{attribute 'global_init_slot' := '40510'}
VAR_GLOBAL
  LblPlt_Facade                                            :FB_BA_Label:=( sObjName:='FAS', sDescr:='Fassade');
  LblPlt_Natural_smoke_extraction                          :FB_BA_Label:=( sObjName:='NRA', sDescr:='Natürlicher Rauchabzug');
  LblPlt_Doors_gates_sluices                               :FB_BA_Label:=( sObjName:='TUE', sDescr:='Türen, Tore, Schleusen');
  LblPlt_Smoke_and_heat_extraction_system                  :FB_BA_Label:=( sObjName:='RWA', sDescr:='Rauch- und Wärmeabzugsanlage');
  LblPlt_Sunlight_protection                               :FB_BA_Label:=( sObjName:='SON', sDescr:='Sonnenschutzanlage');
// 411 Abwasseranlagen
  LblPlt_Separator_facility                                :FB_BA_Label:=( sObjName:='ABS', sDescr:='Abscheideranlage');
  LblPlt_Lifting_system                                    :FB_BA_Label:=( sObjName:='HBA', sDescr:='Hebeanlage');
  LblPlt_Neutralisation_plant                              :FB_BA_Label:=( sObjName:='NEU', sDescr:='Neutralisationsanlage');
// 412 Wasseranlagen
  LblPlt_Trace_heating                                     :FB_BA_Label:=( sObjName:='BGH', sDescr:='Begleitheizung');
  LblPlt_Process_water                                     :FB_BA_Label:=( sObjName:='BTW', sDescr:='Betriebswasser');
  LblPlt_Well_water                                        :FB_BA_Label:=( sObjName:='BWA', sDescr:='Brunnenwasser');
  LblPlt_Dispensing_installation                           :FB_BA_Label:=( sObjName:='DOS', sDescr:='Dosieranlage');
  LblPlt_Pressure_booster_system                           :FB_BA_Label:=( sObjName:='DEA', sDescr:='Druckerhöhungsanlage');
  LblPlt_Softening_unit                                    :FB_BA_Label:=( sObjName:='EHA', sDescr:='Enthärtungsanlage');
// Trinkwasser
  LblPlt_Drinking_water_heating_system                     :FB_BA_Label:=( sObjName:='TWE', sDescr:='Trinkwassererwärmungsanlage');
  LblPlt_Reverse_osmosis_system                            :FB_BA_Label:=( sObjName:='UKO', sDescr:='Umkehrosmoseanlage');
  LblPlt_Desalination_plant                                :FB_BA_Label:=( sObjName:='VEA', sDescr:='Vollentsalzungsanlage');
// 421 Wärmeerzeugungsanlagen
  LblPlt_BHKW                                              :FB_BA_Label:=( sObjName:='BHK', sDescr:='BHKW');
  LblPlt_Electric_heating                                  :FB_BA_Label:=( sObjName:='EHZ', sDescr:='Elektroheizung');
  LblPlt_District_heating_transfer                         :FB_BA_Label:=( sObjName:='FWÜ', sDescr:='Fernwärmeübergabe');
// Geothermieanlage
  LblPlt_Boiler                                            :FB_BA_Label:=( sObjName:='KES', sDescr:='Kessel');
  LblPlt_Clean_steam_generation                            :FB_BA_Label:=( sObjName:='RDE', sDescr:='Reindampferzeugung');
  LblPlt_Solar_power_system                                :FB_BA_Label:=( sObjName:='SOL', sDescr:='Solaranlage');
  LblPlt_Heating_pump                                      :FB_BA_Label:=( sObjName:='WPU', sDescr:='Wärmepumpe');
// 422 Wärmeverteilnetze
  LblPlt_Pressure_maintenance                              :FB_BA_Label:=( sObjName:='DHG', sDescr:='Druckhaltung');
  LblPlt_Heating_circuit                                   :FB_BA_Label:=( sObjName:='HZK', sDescr:='Heizkreis');
  LblPlt_Heating                                           :FB_BA_Label:=( sObjName:='HZG', sDescr:='Heizung');
  LblPlt_Back_feed_system                                  :FB_BA_Label:=( sObjName:='NSA', sDescr:='Nachspeiseanlage');
  LblPlt_Buffer                                            :FB_BA_Label:=( sObjName:='PFS', sDescr:='Pufferspeicher');
  LblPlt_Heat_distribution_network                         :FB_BA_Label:=( sObjName:='WVN', sDescr:='Wärmeverteilnetz');
  LblPlt_Heat_exchanger                                    :FB_BA_Label:=( sObjName:='WTR', sDescr:='Wärmeüberträger');
// 423 Raumheizflächen
  LblPlt_Concrete_core_activation                          :FB_BA_Label:=( sObjName:='BKA', sDescr:='Betonkernaktivierung');
  LblPlt_Overhead_heating                                  :FB_BA_Label:=( sObjName:='DHZ', sDescr:='Deckenheizung');
  LblPlt_Ceiling_radiator_panels                           :FB_BA_Label:=( sObjName:='DSP', sDescr:='Deckenstrahlplatten');
  LblPlt_Facade_heating                                    :FB_BA_Label:=( sObjName:='FAH', sDescr:='Fassadenheizung');
  LblPlt_Panel_heating                                     :FB_BA_Label:=( sObjName:='FLH', sDescr:='Flächenheizung');
  LblPlt_Underfloor_heating                                :FB_BA_Label:=( sObjName:='FBH', sDescr:='Fußbodenheizung');
  LblPlt_Heated_chilled_ceiling                            :FB_BA_Label:=( sObjName:='HKD', sDescr:='Heiz-/Kühldecke');
  LblPlt_Static_heating                                    :FB_BA_Label:=( sObjName:='STH', sDescr:='Statische Heizung');
// 430 Lufttechnische Anlagen
  LblPlt_Extract_air_system                                :FB_BA_Label:=( sObjName:='ABA', sDescr:='Abluftanlage');
  LblPlt_Roof_air_heater                                   :FB_BA_Label:=( sObjName:='DLH', sDescr:='Deckenlufterhitzer');
  LblPlt_Circulatory_system                                :FB_BA_Label:=( sObjName:='KVS', sDescr:='Kreislaufverbundsystem');
  LblPlt_Air_processing_unit                               :FB_BA_Label:=( sObjName:='LAZ', sDescr:='Luftaufbereitungszentrale');
  LblPlt_Mechanical_smoke_extraction_system                :FB_BA_Label:=( sObjName:='MRA', sDescr:='Maschinelle Rauchabzugsanlage');
  LblPlt_Smoke_pressure_system                             :FB_BA_Label:=( sObjName:='RDA', sDescr:='Rauchdruckanlage');
  LblPlt_Air_handling_unit                                 :FB_BA_Label:=( sObjName:='RLT', sDescr:='Raumlufttechnik');
  LblPlt_Partial_air_conditioning_system                   :FB_BA_Label:=( sObjName:='TKA', sDescr:='Teilklimaanlage');
  LblPlt_Air_curtain_system                                :FB_BA_Label:=( sObjName:='TLS', sDescr:='Türluftschleieranlage');
  LblPlt_Recirculating_air_system                          :FB_BA_Label:=( sObjName:='ULA', sDescr:='Umluftanlage');
  LblPlt_Full_air_conditioning_system                      :FB_BA_Label:=( sObjName:='VKA', sDescr:='Vollklimaanlage');
  LblPlt_Heat_recovery_system                              :FB_BA_Label:=( sObjName:='WRG', sDescr:='Wärmerückgewinnungssystem');
  LblPlt_Intake_air_system                                 :FB_BA_Label:=( sObjName:='ZUA', sDescr:='Zuluftanlage');
  LblPlt_Smoke_extraction_system                           :FB_BA_Label:=( sObjName:='ERA', sDescr:='Entrauchungsanlage');
// 434 Kälteanlagen
  LblPlt_Remote_cooling_transfer                           :FB_BA_Label:=( sObjName:='FKÜ', sDescr:='Fernkälteübergabe');
  LblPlt_Cooling                                           :FB_BA_Label:=( sObjName:='KAE', sDescr:='Kälte');
  LblPlt_Cooling_circuit                                   :FB_BA_Label:=( sObjName:='KKR', sDescr:='Kältekreis');
  LblPlt_Cooling_distribution_network                      :FB_BA_Label:=( sObjName:='KVN', sDescr:='Kälteverteilnetz');
  LblPlt_Cold_water_generation                             :FB_BA_Label:=( sObjName:='KWE', sDescr:='Kaltwassererzeugung');
  LblPlt_Electrical_cabinet_cooling                        :FB_BA_Label:=( sObjName:='KVE', sDescr:='Kühlung Schaltschrank ');
  LblPlt_Cooling_storage                                   :FB_BA_Label:=( sObjName:='KSP', sDescr:='Kältespeicher');
  LblPlt_Chilled_ceiling                                   :FB_BA_Label:=( sObjName:='KÜD', sDescr:='Kühldecke');
  LblPlt_Re_cooling_plant                                  :FB_BA_Label:=( sObjName:='RKW', sDescr:='Rückkühlwerk');
// 441 Hoch- und Mittelspannungsanlagen
  LblPlt_Switchgear                                        :FB_BA_Label:=( sObjName:='STA', sDescr:='Schaltanlagen');
  LblPlt_Transformer                                       :FB_BA_Label:=( sObjName:='TRF', sDescr:='Transformator');
  LblPlt_Medium_voltage_system                             :FB_BA_Label:=( sObjName:='MSA', sDescr:='Mittelspannungsanlage');
  LblPlt_Compensation_system                               :FB_BA_Label:=( sObjName:='KOA', sDescr:='Kompensationsanlage');
  LblPlt_Frequency_converter_system                        :FB_BA_Label:=( sObjName:='FUA', sDescr:='Frequenzumformeranlage');
// 442 Eigenstromversorgungsanlagen
  LblPlt_Emissions_system                                  :FB_BA_Label:=( sObjName:='AGA', sDescr:='Abgasanlage');
  LblPlt_Battery_unit                                      :FB_BA_Label:=( sObjName:='BAT', sDescr:='Batterieanlage');
  LblPlt_Co_generation_unit                                :FB_BA_Label:=( sObjName:='BHK', sDescr:='Blockheizkraftwerk');
  LblPlt_Fuel_supply                                       :FB_BA_Label:=( sObjName:='BRV', sDescr:='Brennstoffversorgung');
  LblPlt_Standby_power_system                              :FB_BA_Label:=( sObjName:='ESA', sDescr:='Ersatzstromanlage');
  LblPlt_Photovoltaic_system                               :FB_BA_Label:=( sObjName:='PVA', sDescr:='Fotovoltaikanlage');
  LblPlt_Uninterruptible_power_supply                      :FB_BA_Label:=( sObjName:='USV', sDescr:='Unterbrechungsfreie Stromversorgung');
// 443 Niederspannungsschaltanlagen
  LblPlt_General_power_supply                              :FB_BA_Label:=( sObjName:='ASV', sDescr:='Allgemeine Stromversorgung');
  LblPlt_Safety_power_supply                               :FB_BA_Label:=( sObjName:='SSV', sDescr:='Sicherheitsstromversorgung');
  LblPlt_Lighting                                          :FB_BA_Label:=( sObjName:='BEL', sDescr:='Beleuchtungsanlage');
  LblPlt_Emergency_lighting                                :FB_BA_Label:=( sObjName:='SIB', sDescr:='Sicherheitsbeleuchtung');
// 451 Telekommunikationsanlagen
  LblPlt_Telecommunications_system                         :FB_BA_Label:=( sObjName:='TEL', sDescr:='Telekommunikationsanlage');
// 452 Such- und Signalanlagen
  LblPlt_Call_signalling_system                            :FB_BA_Label:=( sObjName:='LRA', sDescr:='Lichtrufanlage');
  LblPlt_Door_intercom_and_door_opener_system              :FB_BA_Label:=( sObjName:='TÜA', sDescr:='Türsprech- und -öffneranlage');
  LblPlt_Paging_system                                     :FB_BA_Label:=( sObjName:='PRA', sDescr:='Personenrufanlage');
// 453 Zeitdienstanlagen
  LblPlt_Clock_and_time_recording_system                   :FB_BA_Label:=( sObjName:='ZEA', sDescr:='Uhren- und Zeiterfassungsanlage');
// 454 Elektroakustische Anlagen
  LblPlt_Electro_acoustic_sound_systems                    :FB_BA_Label:=( sObjName:='ELA', sDescr:='Elektroakustische Anl. , Beschallung');
  LblPlt_Conference_and_interpreting_equipment             :FB_BA_Label:=( sObjName:='KDA', sDescr:='Konferenz- und Dolmetscheranlage');
  LblPlt_Intercom_system                                   :FB_BA_Label:=( sObjName:='GSA', sDescr:='Gegensprechanlage');
  LblPlt_Voice_alarm_system                                :FB_BA_Label:=( sObjName:='SAA', sDescr:='Sprachalarmierungsanlage');
  LblPlt_Intercommunication_systems                        :FB_BA_Label:=( sObjName:='WSA', sDescr:='Wechselsprechanlagen');
// 455 Fernseh- und Antennenanlagen
  LblPlt_Television_system                                 :FB_BA_Label:=( sObjName:='TVA', sDescr:='Fernsehanlage');
  LblPlt_Transmitting_and_receiving_antenna_system         :FB_BA_Label:=( sObjName:='SEA', sDescr:='Sende- und Empfangsantennenanlage');
  LblPlt_BOS_radio_system                                  :FB_BA_Label:=( sObjName:='BOS', sDescr:='BOS-Funkanlage');
// 456 Gefahrenmelde- und Alarmanlagen
  LblPlt_Fire_detection_and_alarm_system                   :FB_BA_Label:=( sObjName:='BMA', sDescr:='Brandmeldeanlage');
  LblPlt_Carbon_monoxide_warning_system                    :FB_BA_Label:=( sObjName:='COW', sDescr:='CO-Warnanlage');
  LblPlt_Burglar_alarm_system                              :FB_BA_Label:=( sObjName:='EMA', sDescr:='Einbruchmeldeanlage');
  LblPlt_Fire_control_panel                                :FB_BA_Label:=( sObjName:='FWT', sDescr:='Feuerwehrtableau');
  LblPlt_Escape_route_protection_system                    :FB_BA_Label:=( sObjName:='FWS', sDescr:='Fluchtwegsicherungsanlage');
  LblPlt_Hazard_detection_system                           :FB_BA_Label:=( sObjName:='GMA', sDescr:='Gefahrenmeldeanlage');
  LblPlt_Gas_warning_system                                :FB_BA_Label:=( sObjName:='GWA', sDescr:='Gaswarnanlage');
  LblPlt_Smoke_aspiration_system                           :FB_BA_Label:=( sObjName:='RAS', sDescr:='Rauchansaugsystem');
  LblPlt_Room_observation_system                           :FB_BA_Label:=( sObjName:='RBA', sDescr:='Raumbeobachtungsanlage');
  LblPlt_Robbery_alarm_system                              :FB_BA_Label:=( sObjName:='ÜFA', sDescr:='Überfallmeldeanlage');
  LblPlt_Guard_control_system                              :FB_BA_Label:=( sObjName:='WKA', sDescr:='Wächterkontrollanlage');
  LblPlt_Emergency_call_system                             :FB_BA_Label:=( sObjName:='NOT', sDescr:='Notrufanlage');
  LblPlt_Access_control_system                             :FB_BA_Label:=( sObjName:='ZKS', sDescr:='Zugangskontrollsystem');
// 457 Übertragungsnetze
  LblPlt_Networks_for_the_transmission_voice_text_etc      :FB_BA_Label:=( sObjName:='LAN', sDescr:='Netzw.  Daten, Sprache, Text etc');
// 459 Fernmelde- und informationstechnische Anlagen, Sonstiges
  LblPlt_Remote_control_systems                            :FB_BA_Label:=( sObjName:='FWA', sDescr:='Fernwirkanlagen');
  LblPlt_Parking_guidance_systems                          :FB_BA_Label:=( sObjName:='PLS', sDescr:='Parkleitsysteme');
// 460 Förderanlagen
  LblPlt_File_transportation_systems                       :FB_BA_Label:=( sObjName:='ATA', sDescr:='Aktentransportanlagen');
  LblPlt_Lift                                              :FB_BA_Label:=( sObjName:='AUF', sDescr:='Aufzug');
  LblPlt_Inspection_systems                                :FB_BA_Label:=( sObjName:='BFA', sDescr:='Befahranlagen');
  LblPlt_Moving_walkways                                   :FB_BA_Label:=( sObjName:='FST', sDescr:='Fahrsteige');
  LblPlt_Escalators                                        :FB_BA_Label:=( sObjName:='FTR', sDescr:='Fahrtreppen');
  LblPlt_External_lifts                                    :FB_BA_Label:=( sObjName:='FSA', sDescr:='Fassadenaufzüge');
  LblPlt_Baggage_conveyor_system                           :FB_BA_Label:=( sObjName:='GFA', sDescr:='Gepäckförderanlage');
  LblPlt_Pneumatic_delivery_systems                        :FB_BA_Label:=( sObjName:='RPA', sDescr:='Rohrpostanlagen');
  LblPlt_Goods_transportation_facilities                   :FB_BA_Label:=( sObjName:='WTA', sDescr:='Warentransportanlagen');
// 470 Nutzerspezifische Anlagen
// 471 Küchentechnische Anlagen
  LblPlt_Small_refrigeration_unit                          :FB_BA_Label:=( sObjName:='KLK', sDescr:='Kleinkälteanlage');
// 472 Wäscherei- und Reinigungsanlagen
  LblPlt_Disinfection_unit                                 :FB_BA_Label:=( sObjName:='DES', sDescr:='Desinfektionsanlage');
  LblPlt_Cleaning_unit                                     :FB_BA_Label:=( sObjName:='REA', sDescr:='Reinigungsanlage');
  LblPlt_Sterilisation_systems                             :FB_BA_Label:=( sObjName:='STR', sDescr:='Sterilisationseinrichtungen');
  LblPlt_Water_treatment_system                            :FB_BA_Label:=( sObjName:='WAA', sDescr:='Wasseraufbereitungsanlage');
  LblPlt_Laundry_system                                    :FB_BA_Label:=( sObjName:='WÄA', sDescr:='Wäschereianlage');
// 473 Medienversorgungsanlagen
  LblPlt_Compressed_air_supply_system                      :FB_BA_Label:=( sObjName:='DRL', sDescr:='Druckluftversorgungsanlage');
  LblPlt_Pressure_regulator_unit                           :FB_BA_Label:=( sObjName:='DRA', sDescr:='Druckregelanlage');
  LblPlt_Media_supply_system                               :FB_BA_Label:=( sObjName:='MVA', sDescr:='Medienversorgungsanlage');
  LblPlt_Medical_and_technical_gases                       :FB_BA_Label:=( sObjName:='MTG', sDescr:='Medizinische und technische Gase');
  LblPlt_Vacuum_unit                                       :FB_BA_Label:=( sObjName:='VAK', sDescr:='Vakuumanlage');
// 474 Medizin- und labortechnische Anlagen
  LblPlt_Medical_technical_plant                           :FB_BA_Label:=( sObjName:='MED', sDescr:='Medizintechnische Anlagen');
  LblPlt_Medical_gas_supply                                :FB_BA_Label:=( sObjName:='MGV', sDescr:='Medizinische Gasversorgung');
  LblPlt_Laboratory_equipment                              :FB_BA_Label:=( sObjName:='LAB', sDescr:='Labortechnische Anlagen (allgemein)');
// 475 Feuerlöschanlagen
  LblPlt_Fire_extinguisher                                 :FB_BA_Label:=( sObjName:='FLA', sDescr:='Feuerlöschanlage');
  LblPlt_Gas_extinguishing_system                          :FB_BA_Label:=( sObjName:='GLA', sDescr:='Gaslöschanlage');
  LblPlt_Fire_extinguishing_system                         :FB_BA_Label:=( sObjName:='LÖS', sDescr:='Löschanlage (allgemein)');
  LblPlt_Mist_extinguishing_system                         :FB_BA_Label:=( sObjName:='NLA', sDescr:='Nebellöschanlage');
  LblPlt_NOX_system                                        :FB_BA_Label:=( sObjName:='NOX', sDescr:='NOX-Anlage');
  LblPlt_Sprinkler_system                                  :FB_BA_Label:=( sObjName:='SPR', sDescr:='Sprinkleranlage');
  LblPlt_Wall_hydrant_system                               :FB_BA_Label:=( sObjName:='WHA', sDescr:='Wandhydrantenanlage');
// 478 Entsorgungsanlagen
  LblPlt_Waste_disposal_system                             :FB_BA_Label:=( sObjName:='AEA', sDescr:='Abfallentsorgungsanlage');
  LblPlt_Media_disposal_system                             :FB_BA_Label:=( sObjName:='MEA', sDescr:='Medienentsorgungsanlage');
  LblPlt_Vacuum_cleaning_systems                           :FB_BA_Label:=( sObjName:='SSA', sDescr:='Staubsauganlagen');
// 480 Gebäudeautomation
  LblPlt_Automation_control_equipment                      :FB_BA_Label:=( sObjName:='ASP', sDescr:='Automationsschwerpunkt');
  LblPlt_Weather_station                                   :FB_BA_Label:=( sObjName:='WET', sDescr:='Wetterstation');
  LblPlt_Management_and_operating_equipment                :FB_BA_Label:=( sObjName:='MBE', sDescr:='Management- und Bedieneinrichtungen');
  LblPlt_Room_automation                                   :FB_BA_Label:=( sObjName:='RAU', sDescr:='Raumautomation');
  LblPlt_Room_automation_system_distributor                :FB_BA_Label:=( sObjName:='RAV', sDescr:='Raumautomation-Systemverteiler');
  LblPlt_Control_cabinet                                   :FB_BA_Label:=( sObjName:='SSK', sDescr:='Schaltschrank');
  LblPlt_Settings                                          :FB_BA_Label:=( sObjName:='ALP', sDescr:='Anlagenparameter');
  LblPlt_EventGroups                                       :FB_BA_Label:=( sObjName:='ERG', sDescr:='Meldeklassen');
  LblPlt_Global_Building_Data                              :FB_BA_Label:=( sObjName:='GGL', sDescr:='Globale Gebäudedaten');
// 540 Technische Anlagen in Außenanlagen
  LblPlt_Rainwater_retention_basin                         :FB_BA_Label:=( sObjName:='RRB', sDescr:='Regenrückhaltebecken');
  LblPlt_Cistern_system                                    :FB_BA_Label:=( sObjName:='ZTA', sDescr:='Zisternenanlage');
END_VAR

// ---- Templates/GVLs/Language/German/TxtEvent_DE.TcGVL
{region '#Template'}
	{attribute 'Version' := '5.0.0.0'}
	{attribute 'Tags' := '"LCID": "1031", "Text": "GVL, Property, Event, Event Message Text, Active Text, Inactive Text"'}
	{attribute 'Tags' := '"LCID": "1033", "Text": "GVL, Property, Event, Event Message Text, Active Text, Inactive Text"'}
	{attribute 'Description' := '"LCID": "1031", "Text": "Textliste Properties Event Message Text, Active Text, Inactive Text"'}
	{attribute 'Description' := '"LCID": "1033", "Text": "Text list Properties Event Message Text, Active Text, Inactive Text"'}
{endregion}

{attribute 'global_init_slot' := '40510'}
VAR_GLOBAL
  txtEvent_No                                                :T_BA_StateText:='Nein';
  txtEvent_Yes                                               :T_BA_StateText:='Ja';
  txtEvent_Auto                                              :T_BA_StateText:='Automatik';
  txtEvent_Manual                                            :T_BA_StateText:='Hand';
  txtEvent_Off                                               :T_BA_StateText:='Aus';
  txtEvent_On                                                :T_BA_StateText:='Ein';
  txtEvent_Opened                                            :T_BA_StateText:='Geöffnet';
  txtEvent_Closed                                            :T_BA_StateText:='Geschlossen';
  txtEvent_Open                                              :T_BA_StateText:='Auf';
  txtEvent_Close                                             :T_BA_StateText:='Zu';
  txtEvent_Step1                                             :T_BA_StateText:='Stufe 1 ';
  txtEvent_Step2                                             :T_BA_StateText:='Stufe 2';
  txtEvent_Step3                                             :T_BA_StateText:='Stufe 3';
  txtEvent_Step4                                             :T_BA_StateText:='Stufe 4';
  txtEvent_Step5                                             :T_BA_StateText:='Stufe 5';
  txtEvent_Step6                                             :T_BA_StateText:='Stufe 6';
  txtEvent_Step7                                             :T_BA_StateText:='Stufe 7';
  txtEvent_Step8                                             :T_BA_StateText:='Stufe 8';
  txtEvent_Released                                          :T_BA_StateText:='Freigegeben';
  txtEvent_Inactive                                          :T_BA_StateText:='Inaktiv';
  txtEvent_Active                                            :T_BA_StateText:='Aktiv';
  txtEvent_Normal                                            :T_BA_StateText:='Normal';
  txtEvent_Offnormal                                         :T_BA_StateText:='Unnormal';
  txtEvent_Alert                                             :T_BA_StateText:='Alarm';
  txtEvent_Disturb                                           :T_BA_StateText:='Störung';
  txtEvent_Error                                             :T_BA_StateText:='Fehler ';
  txtEvent_Triggered                                         :T_BA_StateText:='Ausgelöst';
  txtEvent_Maintenace                                        :T_BA_StateText:='Wartung';
  txtEvent_Exceeded                                          :T_BA_StateText:='Überschritten';
  txtEvent_Monitoring                                        :T_BA_StateText:='Überwachung';
  txtEvent_Protection                                        :T_BA_StateText:='Schutzbetrieb';
  txtEvent_Economy                                           :T_BA_StateText:='Economy';
  txtEvent_PreComfort                                        :T_BA_StateText:='Pre-Comfort';
  txtEvent_Comfort                                           :T_BA_StateText:='Comfort';
  txtEvent_Reached                                           :T_BA_StateText:='erreicht';
  txtEvent_NotReached                                        :T_BA_StateText:='nicht erreicht';
  txtEvent_None                                              :T_BA_StateText:='""';
  txtEvent_EmergencyStop                                     :T_BA_StateText:='Notaus';
  txtEvent_Frost                                             :T_BA_StateText:='Frost';
  txtEvent_SmokeExtraction_P                                 :T_BA_StateText:='Entrauchung mit Zu- und Abluft';
  txtEvent_SmokeExtractionSupplyAir                          :T_BA_StateText:='Entrauchung Zuluft';
  txtEvent_SmokeExtractionExtractAir                         :T_BA_StateText:='Entrauchung Abluft';
  txtEvent_CoolDownProtection                                :T_BA_StateText:='Auskühlschutz';
  txtEvent_OverHeatingProtection                             :T_BA_StateText:='Überhitzungsschutz';
  txtEvent_Fire                                              :T_BA_StateText:='Brandalarm';
  txtEvent_NightCooling                                      :T_BA_StateText:='Nachtkühlung';
  txtEvent_ForcedVentilation                                 :T_BA_StateText:='Zwangsbelüftung';
  txtEvent_CentralSwitchOff                                  :T_BA_StateText:='Zentralaus';
  txtEvent_Locked                                            :T_BA_StateText:='verriegelt';
  txtEvent_Contaminated                                      :T_BA_StateText:='verschmutzt';
  txtEvent_Stop                                              :T_BA_StateText:='Stop';
  txtEvent_Critical                                          :T_BA_StateText:='kritisch';
  txtEvent_UnCiritical                                       :T_BA_StateText:='unkritisch';
  txtEvent_Average                                           :T_BA_StateText:='Mittelwert';
  txtEvent_HeatCool                                          :T_BA_StateText:='Heiz/Kühl';
  txtEvent_AverageHeatCool                                   :T_BA_StateText:='Mittelwert Heizen/Kühlen';
  txtEvent_Direction                                         :T_BA_StateText:='Wirksinn';
  txtEvent_Default                                           :T_BA_StateText:='Standard';
  txtEvent_Cleaning                                          :T_BA_StateText:='Gebaeudereinigung';
  txtEvent_Nightwatch                                        :T_BA_StateText:='Nachtwaechter';
  txtEvent_SupplyAirTControlReheater                         :T_BA_StateText:='Zulufttemperaturregelung Nacherhitzer';
  txtEvent_SupplyAirTControlPreheater                        :T_BA_StateText:='Zulufttemperaturregelung Vorerhitzer';
  txtEvent_SupplyAirTControlERC                              :T_BA_StateText:='Zulufttemperaturregelung WRG';
  txtEvent_SupplyAirTControlMix                              :T_BA_StateText:='Zulufttemperaturregelung Mischluft';
  txtEvent_SupplyAirTControlCooler                           :T_BA_StateText:='Zulufttemperaturregelung Kühler';
  txtEvent_SupplyAirXControlCooler                           :T_BA_StateText:='Zuluftfeuchtereglung Kühler';
  txtEvent_SupplyAirXControlHumf                             :T_BA_StateText:='Zuluftfeuchtereglung Befeuchter';
  txtEvent_PreRinse                                          :T_BA_StateText:='Vorspülen';
  txtEvent_DamperOpen                                        :T_BA_StateText:='Klappen Auf';
  txtEvent_SupplyAirFan                                      :T_BA_StateText:='Zuluft Ventilator';
  txtEvent_ExtractAirFan                                     :T_BA_StateText:='Abluft Ventilator';
  txtEvent_EnableTemperatureControl                          :T_BA_StateText:='Freigabe Temperatur Regelung';
  txtEvent_EnableTemperatureSequenceLink                     :T_BA_StateText:='Freigabe Temperatur Sequenz Steuerung';
  txtEvent_EnableHumidityControl                             :T_BA_StateText:='Freigabe Feuchte Regelung';
  txtEvent_EnableHumiditySequenceLink                        :T_BA_StateText:='Freigabe Feuchte Sequenz Steuerung';
  txtEvent_ReleaseLimitMonitoring                            :T_BA_StateText:='Freigabe Grenzwertüberwachung';
  txtEvent_Reheater                                          :T_BA_StateText:='Nacherhitzer';
  txtEvent_Preheater                                         :T_BA_StateText:='Vorerhitzer';
  txtEvent_MixedAir                                          :T_BA_StateText:='Mischluft';
  txtEvent_EnergyRecovery                                    :T_BA_StateText:='Energierückgewinnung';
  txtEvent_Cooler                                            :T_BA_StateText:='Kühler';
  txtEvent_Humidifier                                        :T_BA_StateText:='Befeuchter';
  txtEvent_Dehumidifier                                      :T_BA_StateText:='Entfeuchter';
  txtEvent_DamperExhaustAir                                  :T_BA_StateText:='Fortluftklappe';
  txtEvent_DamperOutsideAir                                  :T_BA_StateText:='Aussenluftklappe';
END_VAR

// ---- Templates/GVLs/Language/German/TxtTrade_DE.TcGVL
{region '#Template'}
	{attribute 'Version' := '5.0.0.0'}
	{attribute 'Tags' := '"LCID": "1031", "Text": "GVL, DPAD, Trades, ObjectName, Description"'}
	{attribute 'Tags' := '"LCID": "1033", "Text": "GVL, DPAD, Trades, ObjectName, Description"'}
	{attribute 'Description' := '"LCID": "1031", "Text": "Textliste Gewerke"'}
	{attribute 'Description' := '"LCID": "1033", "Text": "Text list trades"'}
{endregion}

{attribute 'global_init_slot' := '40510'}
VAR_GLOBAL
  TxtTrade_Doors_gates_windows_sun_protection_sObjectName                :T_BA_StateText:='TTF';
  TxtTrade_Doors_gates_windows_sun_protection_sDescription                :T_BA_StateText:='Türen, Tore, Fenster, Sonnenschutz';
  TxtTrade_Sewage_water_and_gas_plants_sObjectName                       :T_BA_StateText:='GWA';
  TxtTrade_Sewage_water_and_gas_plants_sDescription                       :T_BA_StateText:='Abwasser-, Wasser-, Gasanlagen';
  TxtTrade_Heat_supply_systems_sObjectName                               :T_BA_StateText:='HZG';
  TxtTrade_Heat_supply_systems_sDescription                               :T_BA_StateText:='Wärmeversorgungsanlagen';
  TxtTrade_Air_conditioning_sObjectName                                  :T_BA_StateText:='LTA';
  TxtTrade_Air_conditioning_sDescription                                  :T_BA_StateText:='Lufttechnische Anlagen';
  TxtTrade_Refrigeration_systems_sObjectName                             :T_BA_StateText:='KAE';
  TxtTrade_Refrigeration_systems_sDescription                             :T_BA_StateText:='Kälteanlagen';
  TxtTrade_High_voltage_systems_sObjectName                              :T_BA_StateText:='ELT';
  TxtTrade_High_voltage_systems_sDescription                              :T_BA_StateText:='Starkstromanlagen';
  TxtTrade_Telecommunication_and_information_technology_sObjectName      :T_BA_StateText:='FIA';
  TxtTrade_Telecommunication_and_information_technology_sDescription      :T_BA_StateText:='Fernm.- und informationstech. Anlagen';
  TxtTrade_Hazard_detection_and_alarm_systems_sObjectName                :T_BA_StateText:='GMA';
  TxtTrade_Hazard_detection_and_alarm_systems_sDescription                :T_BA_StateText:='Gefahrenmelde- und Alarmanlagen';
  TxtTrade_Conveyors_sObjectName                                         :T_BA_StateText:='FTA';
  TxtTrade_Conveyors_sDescription                                         :T_BA_StateText:='Förderanlagen';
  TxtTrade_Kitchen_technology_systems_sObjectName                        :T_BA_StateText:='KTA';
  TxtTrade_Kitchen_technology_systems_sDescription                        :T_BA_StateText:='Küchentechnische Anlagen';
  TxtTrade_Laundry_and_cleaning_systems_sObjectName                      :T_BA_StateText:='WAR';
  TxtTrade_Laundry_and_cleaning_systems_sDescription                      :T_BA_StateText:='Wäscherei- und Reinigungsanlagen';
  TxtTrade_Media_supply_systems_sObjectName                              :T_BA_StateText:='MVA';
  TxtTrade_Media_supply_systems_sDescription                              :T_BA_StateText:='Medienversorgungsanlagen';
  TxtTrade_Medical_and_laboratory_equipment_sObjectName                  :T_BA_StateText:='MED';
  TxtTrade_Medical_and_laboratory_equipment_sDescription                  :T_BA_StateText:='Medizin- und labortechnische Anlagen';
  TxtTrade_Fire_extinguishing_systems_sObjectName                        :T_BA_StateText:='FLA';
  TxtTrade_Fire_extinguishing_systems_sDescription                        :T_BA_StateText:='Feuerlöschanlagen';
  TxtTrade_Bathing_facilities_sObjectName                                :T_BA_StateText:='BTA';
  TxtTrade_Bathing_facilities_sDescription                                :T_BA_StateText:='Badetechnische Anlagen';
  TxtTrade_Process_heating_cooling_and_air_systems_sObjectName           :T_BA_StateText:='PRO';
  TxtTrade_Process_heating_cooling_and_air_systems_sDescription           :T_BA_StateText:='Prozesswärme-, -kälte- und -luftanlagen';
  TxtTrade_Waste_disposal_facilities_sObjectName                         :T_BA_StateText:='ENT';
  TxtTrade_Waste_disposal_facilities_sDescription                         :T_BA_StateText:='Entsorgungsanlagen';
  TxtTrade_Building_automation_and_control_systems_general_sObjectName   :T_BA_StateText:='GAS';
  TxtTrade_Building_automation_and_control_systems_general_sDescription   :T_BA_StateText:='Gebäudeautomation allgemein';
  TxtTrade_Automation_focal_point_information_focal_point_sObjectName    :T_BA_StateText:='ASP';
  TxtTrade_Automation_focal_point_information_focal_point_sDescription    :T_BA_StateText:='Automationsschwerpunkt';
  TxtTrade_Room_automation_sObjectName                                   :T_BA_StateText:='RAU';
  TxtTrade_Room_automation_sDescription                                   :T_BA_StateText:='Raumautomation';
  TxtTrade_Outdoor_devices_sObjectName                                   :T_BA_StateText:='AUG';
  TxtTrade_Outdoor_devices_sDescription                                   :T_BA_StateText:='Außengeräte';
END_VAR

// ---- Templates/GVLs/LblComp.TcGVL
{region '#Template'}
	{attribute 'Version' := '5.1.0.0'}
	{attribute 'Tags' := '"LCID": "1031", "Text": "GVL, Kompositionen von Labels für Sonderfunktionen"'}
	{attribute 'Tags' := '"LCID": "1033", "Text": "GVL, LabelComposition for Secial Functions"'}
	{attribute 'Description' := '"LCID": "1031", "Text": "Label Kompositionen"'}
	{attribute 'Description' := '"LCID": "1033", "Text": "Label composition"'}
{endregion}

{attribute 'global_init_slot' := '40520'}
VAR_GLOBAL
	LblComp_Project								:FB_BA_Label2x:=(iAggregate:=LblAgg_AutomationStationEquipment,	iFunction:=LblCTL_BACnetDevice);
	
	//     Composition of 2 Labels
	//     479 User-specific system, weather station 
	LblComp_Wth_RainSensor						:FB_BA_Label2x:=(iAggregate:=LblAgg_RainSensor,			iFunction:=LblFun_OperationalMessage);
	LblComp_Wth_WeatherStation					:FB_BA_Label2x:=(iAggregate:=LblAgg_WeatherStation,		iFunction:=LblFun_Fault);
												
	LblComp_Wth_TemperatureOutside				:FB_BA_Label2x:=(iAggregate:=LblAgg_TemperatureOutside,	iFunction:=LblFun_MeasuredValue);
	LblComp_Wth_TemperatureDewPoint				:FB_BA_Label2x:=(iAggregate:=LblAgg_TemperatureDewPoint,iFunction:=LblFun_MeasuredValue);
	LblComp_Wth_PressureAbsolute				:FB_BA_Label2x:=(iAggregate:=LblAgg_PressureAbsolute,	iFunction:=LblFun_MeasuredValue);
	LblComp_Wth_PressureRelative				:FB_BA_Label2x:=(iAggregate:=LblAgg_PressureRelative,	iFunction:=LblFun_MeasuredValue);
	LblComp_Wth_AbsoluteHumidityOutsideAir		:FB_BA_Label2x:=(iAggregate:=LblAgg_AbsoluteHumidityOutsideAir,iFunction:=LblFun_MeasuredValue);
	LblComp_Wth_RelativeHumidityOutsideAir		:FB_BA_Label2x:=(iAggregate:=LblAgg_RelativeHumidityOutsideAir,iFunction:=LblFun_MeasuredValue);
	LblComp_Wth_Brightness						:FB_BA_Label2x:=(iAggregate:=LblAgg_Brightness,			iFunction:=LblFun_MeasuredValue);
	LblComp_Wth_Dawn							:FB_BA_Label2x:=(iAggregate:=LblAgg_Dawn,				iFunction:=LblFun_MeasuredValue);
	LblComp_Wth_SolarRadiation					:FB_BA_Label2x:=(iAggregate:=LblAgg_SolarRadiation,		iFunction:=LblFun_MeasuredValue);
	LblComp_Wth_WindDirection					:FB_BA_Label2x:=(iAggregate:=LblAgg_WindDirection,		iFunction:=LblFun_MeasuredValue);
	LblComp_Wth_WindSpeed						:FB_BA_Label2x:=(iAggregate:=LblAgg_WindSpeed,			iFunction:=LblFun_MeasuredValue);
	LblComp_Wth_GeoLatitude						:FB_BA_Label2x:=(iAggregate:=LblAgg_GeoLatitude,		iFunction:=LblFun_MeasuredValue);
	LblComp_Wth_GeoLongitude					:FB_BA_Label2x:=(iAggregate:=LblAgg_GeoLongitude,		iFunction:=LblFun_MeasuredValue);
	LblComp_Wth_SunAzimuth						:FB_BA_Label2x:=(iAggregate:=LblAgg_SunAzimuth,			iFunction:=LblFun_MeasuredValue);
	LblComp_Wth_SunElevation					:FB_BA_Label2x:=(iAggregate:=LblAgg_SunElevation,		iFunction:=LblFun_MeasuredValue);
	
	LblComp_Wth_WeatherStationReset       		:FB_BA_Label2x:=(iAggregate:=LblAgg_WeatherStationReset,iFunction:=LblFun_SwitchingCommand);
	LblComp_Wth_WeatherStationCommReset   		:FB_BA_Label2x:=(iAggregate:=LblAgg_WeatherStationCommReset,iFunction:=LblFun_SwitchingCommand);
	LblComp_Wth_WeatherStationComm        		:FB_BA_Label2x:=(iAggregate:=LblAgg_WeatherStationComm,	iFunction:=LblFun_Fault);  


	// Temperature // Temperatur
	LblComp_TempExtA_MV        			   		:FB_BA_Label2x:=(iAggregate:=LblAgg_TemperatureExtractAir,		iFunction:=LblFun_MeasuredValue);  
	LblComp_TempExhA_MV        			   		:FB_BA_Label2x:=(iAggregate:=LblAgg_TemperatureExhaustAir,		iFunction:=LblFun_MeasuredValue);  
	LblComp_TempOuA_MV        			   		:FB_BA_Label2x:=(iAggregate:=LblAgg_TemperatureOutside,			iFunction:=LblFun_MeasuredValue);  
	LblComp_TempRmA_MV        			   		:FB_BA_Label2x:=(iAggregate:=LblAgg_TemperatureRoomAir,			iFunction:=LblFun_MeasuredValue);  
	LblComp_TempSuA_MV        			   		:FB_BA_Label2x:=(iAggregate:=LblAgg_TemperatureSupplyAir,		iFunction:=LblFun_MeasuredValue);  
	
	// Relative humidity // Relative Feuchte
	LblComp_RelHumExtA_MV        			   	:FB_BA_Label2x:=(iAggregate:=LblAgg_RelativeHumidityExtractAir,		iFunction:=LblFun_MeasuredValue);  
	LblComp_RelHumExhA_MV        			   	:FB_BA_Label2x:=(iAggregate:=LblAgg_RelativeHumidityExhaustAir,		iFunction:=LblFun_MeasuredValue);  
	LblComp_RelHumOuA_MV        			   	:FB_BA_Label2x:=(iAggregate:=LblAgg_RelativeHumidityOutsideAir,		iFunction:=LblFun_MeasuredValue);  
	LblComp_RelHumRmA_MV        			   	:FB_BA_Label2x:=(iAggregate:=LblAgg_RelativeHumidityRoomHumidity,	iFunction:=LblFun_MeasuredValue);  
	LblComp_RelHumSuA_MV        			   	:FB_BA_Label2x:=(iAggregate:=LblAgg_RelativeHumiditySupplyAir,		iFunction:=LblFun_MeasuredValue);  
	
	// Absolute humidity // Absolute Feuchte
	LblComp_AbsHumExtA_MVC       			   	:FB_BA_Label2x:=(iAggregate:=LblAgg_AbsoluteHumidityExtractAir,	iFunction:=LblFun_MeasuredValueCalculated);  
	LblComp_AbsHumExhA_MVC       			   	:FB_BA_Label2x:=(iAggregate:=LblAgg_AbsoluteHumidityExhaustAir,	iFunction:=LblFun_MeasuredValueCalculated);  
	LblComp_AbsHumOuA_MVC        			   	:FB_BA_Label2x:=(iAggregate:=LblAgg_AbsoluteHumidityOutsideAir,	iFunction:=LblFun_MeasuredValueCalculated);  
	LblComp_AbsHumRmA_MVC        			   	:FB_BA_Label2x:=(iAggregate:=LblAgg_AbsoluteHumidityRoomAir,	iFunction:=LblFun_MeasuredValueCalculated);  
	LblComp_AbsHumSuA_MVC        			   	:FB_BA_Label2x:=(iAggregate:=LblAgg_AbsoluteHumiditySupplyAir,	iFunction:=LblFun_MeasuredValueCalculated);  
	
	// Dew point temperature // Taupunkttemperatur
	LblComp_DewPntExtA_MVC       			   	:FB_BA_Label2x:=(iAggregate:=LblAgg_TemperatureDewPointExtractAir,	iFunction:=LblFun_MeasuredValueCalculated);  
	LblComp_DewPntExhA_MVC       			   	:FB_BA_Label2x:=(iAggregate:=LblAgg_TemperatureDewPointExhaustAir,	iFunction:=LblFun_MeasuredValueCalculated);  
	LblComp_DewPntOuA_MVC        			   	:FB_BA_Label2x:=(iAggregate:=LblAgg_TemperatureDewPointOutsideAir,	iFunction:=LblFun_MeasuredValueCalculated);  
	LblComp_DewPntRmA_MVC        			   	:FB_BA_Label2x:=(iAggregate:=LblAgg_TemperatureDewPointRoomAir,	iFunction:=LblFun_MeasuredValueCalculated);  
	LblComp_DewPntSuA_MVC        			   	:FB_BA_Label2x:=(iAggregate:=LblAgg_TemperatureDewPointSupplyAir,	iFunction:=LblFun_MeasuredValueCalculated);  
	
	// Enthalpy // Enthalpie
	LblComp_EnthalpyExtA_MVC       			   	:FB_BA_Label2x:=(iAggregate:=LblAgg_EnthalpyExtractAir,	iFunction:=LblFun_MeasuredValueCalculated);  
	LblComp_EnthalpyExhA_MVC       			   	:FB_BA_Label2x:=(iAggregate:=LblAgg_EnthalpyExhaustAir,	iFunction:=LblFun_MeasuredValueCalculated);  
	LblComp_EnthalpyOuA_MVC        			   	:FB_BA_Label2x:=(iAggregate:=LblAgg_EnthalpyOutsideAir,	iFunction:=LblFun_MeasuredValueCalculated);  
	LblComp_EnthalpyRmA_MVC        			   	:FB_BA_Label2x:=(iAggregate:=LblAgg_EnthalpyRoomAir,	iFunction:=LblFun_MeasuredValueCalculated);  
	LblComp_EnthalpySuA_MVC        			   	:FB_BA_Label2x:=(iAggregate:=LblAgg_EnthalpySupplyAir,	iFunction:=LblFun_MeasuredValueCalculated);  
	
	// Wet bulp temperature // Feuchtkugeltemperatur
	LblComp_TempWetBulpExtA_MVC       	   		:FB_BA_Label2x:=(iAggregate:=LblAgg_TemperatureWetBulpExtractAir,	iFunction:=LblFun_MeasuredValueCalculated);  
	LblComp_TempWetBulpExhA_MVC       	   		:FB_BA_Label2x:=(iAggregate:=LblAgg_TemperatureWetBulpExhaustAir,	iFunction:=LblFun_MeasuredValueCalculated);  
	LblComp_TempWetBulpOuA_MVC        	   		:FB_BA_Label2x:=(iAggregate:=LblAgg_TemperatureWetBulpOutsideAir,	iFunction:=LblFun_MeasuredValueCalculated);  
	LblComp_TempWetBulpRmA_MVC        	   		:FB_BA_Label2x:=(iAggregate:=LblAgg_TemperatureWetBulpRoomAir,		iFunction:=LblFun_MeasuredValueCalculated);  
	LblComp_TempWetBulpSuA_MVC        	   		:FB_BA_Label2x:=(iAggregate:=LblAgg_TemperatureWetBulpSupplyAir,	iFunction:=LblFun_MeasuredValueCalculated);  
END_VAR

// ---- Templates/GVLs/Site/Site.TcGVL
{region '#Template'}
	{attribute 'Version' := '5.0.1.0'}
	{attribute 'Tags' := '"LCID": "1031", "Text": "GVL, Publisher, Subscriber"'}
	{attribute 'Tags' := '"LCID": "1033", "Text": "GVL, Publisher, Subscriber"'}
	{attribute 'Using' := '"Type": "Template", "URI": "ST_BA_GeneralSettings"'}
	{attribute 'Using' := '"Type": "Template", "URI": "E_BA_EnergyLvlEx"'}
	{attribute 'Using' := '"Type": "Template", "URI": "E_BA_BuildingMode"'}
	{attribute 'Using' := '"Type": "Template", "URI": "ST_BA_BuildingSunBlind"'}
	{attribute 'Using' := '"Type": "Template", "URI": "ST_BA_BuildingAlarms"'}
	{attribute 'Using' := '"Type": "Template", "URI": "ST_BA_WeatherStation"'}
	{attribute 'Using' := '"Type": "Template", "URI": "ST_BA_Facade"'}		 
	{attribute 'Description' := '"LCID": "1031", "Text": "Ams NetId, Subject"'}
	{attribute 'Description' := '"LCID": "1033", "Text": "Ams NetId, Subject"'}
{endregion}

{attribute 'qualified_only'}
VAR_GLOBAL	
	Self_NetId						: T_BA_MedString	:= '127.0.0.1.1.1';
	ACE01_NetId						: T_BA_MedString	:= Self_NetId;
	ACE02_NetId						: T_BA_MedString	:= Self_NetId;
	ACE03_NetId						: T_BA_MedString	:= Self_NetId;
	ACE04_NetId						: T_BA_MedString	:= Self_NetId;
	ACE05_NetId						: T_BA_MedString	:= Self_NetId;
	                            	
	GeneralSettings_Subject			: T_BA_MedString	:= 'GeneralSettings';	
	GeneralSettings_NetId			: T_BA_MedString	:= Self_NetId;	
		                        	
	WeatherStation_Subject			: T_BA_MedString	:= 'WeatherStation';
	WeatherStation_NetId			: T_BA_MedString	:= Self_NetId;
                                	
	FacadeNorth_NetId				: T_BA_MedString	:= ACE01_NetId;
	FacadeNorth_Subject				: T_BA_MedString	:= 'FcdNorth.FacadeSunBlind';
	FacadeEast_NetId				: T_BA_MedString	:= ACE01_NetId;
	FacadeEast_Subject				: T_BA_MedString	:= 'FcdEast.FacadeSunBlind';
	FacadeSouth_NetId				: T_BA_MedString	:= ACE01_NetId;
	FacadeSouth_Subject				: T_BA_MedString	:= 'FcdSouth.FacadeSunBlind';
	FacadeWest_NetId				: T_BA_MedString	:= ACE01_NetId;
	FacadeWest_Subject				: T_BA_MedString	:= 'FcdWest.FacadeSunBlind';
                                	
	Building_NetId					: T_BA_MedString	:= ACE01_NetId;
	BuildingAlarms_Subject			: T_BA_MedString	:= 'BuildingAlarms';
	BuildingMode_Subject			: T_BA_MedString	:= 'BuildingMode';
	BuildingEnergyLevel_Subject		: T_BA_MedString	:= 'BuildingEnergyLevel';
	BuildingSpRmT_Subject			: T_BA_MedString	:= 'BuildingSpRmT';
	BuildingSunProtection_Subject	: T_BA_MedString	:= 'BuildingSunProtection';
	
	
	stGeneralSettings				: ST_BA_GeneralSettings;	// published by FB_BA_Settings	
	bGeneralSettings_Error			: BOOL;	
	eBuildingEnergyLevel			: E_BA_EnergyLvlEx;			// published by FB_BA_BuildingEnergyLevel
	bBuildingEnergyLevel_Error		: BOOL;
	eBuildingMode					: E_BA_BuildingMode;		// published by FB_BA_BuildingMode
	bBuildingMode_Error				: BOOL;
	stBuildingSunBlind				: ST_BA_BuildingSunBlind;	// published by FB_BA_BuildingSunprotection
	bBuildingSunBlind_Error			: BOOL;
	stBuildingAlarms				: ST_BA_BuildingAlarms;		// published by FB_BA_BuildingAlarms
	bBuildingAlarms_Error			: BOOL;
	stWeatherStation				: ST_BA_WeatherStation;		// published by FB_BA_WeatherStation_xxx
	bWeatherStation_Error			: BOOL;
	stFacadeNorthSunBlind			: ST_BA_Facade;				// published by FB_BA_Facade
	bFacadeNorthSunBlind_Error		: BOOL;
	stFacadeEastSunBlind			: ST_BA_Facade;				// published by FB_BA_Facade
	bFacadeEastSunBlind_Error		: BOOL;
	stFacadeSouthSunBlind			: ST_BA_Facade;				// published by FB_BA_Facade
	bFacadeSouthSunBlind_Error		: BOOL;
	stFacadeWestSunBlind			: ST_BA_Facade;				// published by FB_BA_Facade
	bFacadeWestSunBlind_Error		: BOOL;
	stBuildingSpRmT					: ST_BA_SpRmT;				// Published by FB_BA_BuildingSpRmT
	bBuildingSpRmT_Error			: BOOL;
END_VAR

// ---- POUs/MAIN.TcPOU
PROGRAM MAIN
VAR
DPAD		: FB_BA_CarelessDPAD := (
					aIdentifier := [
	(* Level 1 *)		(	eNodeType:=E_BA_NodeType.eBuilding,			sSeparator_ObjectName := '-', 	sSeparator_Description := ' - ',	nIndexDigits := 0),
	(* Level 2 *)		(	eNodeType:=E_BA_NodeType.eFloor,			sSeparator_ObjectName := '-', 	sSeparator_Description := ' - ',	nIndexDigits := 0),
	(* Level 3 *)		(	eNodeType:=E_BA_NodeType.eTrade,			sSeparator_ObjectName := '-', 	sSeparator_Description := ' - ',	nIndexDigits := 0),
	(* Level 4 *)		(	eNodeType:=E_BA_NodeType.ePlant,			sSeparator_ObjectName := '-', 	sSeparator_Description := ' - ',	nIndexDigits := 2),
	(* Level 5 *)		(	eNodeType:=E_BA_NodeType.eAggregate,		sSeparator_ObjectName := '-', 	sSeparator_Description := ' - ',	nIndexDigits := 2),
	(* Level 6 *)		(	eNodeType:=E_BA_NodeType.eFunction,			sSeparator_ObjectName := '-', 	sSeparator_Description := ' - ',	nIndexDigits := 2)
					]
				);				

			
//	Level 1 Gebäude 	
//	Level 1 Building 	
		B			: FB_BA_View := (
						sObjectName		:= 'B',	
						sDescription	:= 'Building B',	
						eDPADMode		:= E_BA_DPADMode.eInclude					
					);     
  
// Level 2 Stockwerk 	->	O01 = Obergeschoss 01, U01 = Untergeschoss 01,  E00 = Ergeschoss
// Level 2 floor ->	F01 = floor 01, B01 = basement 01,  GFL = Ground floor  						
			F01			: FB_BA_View := (
							iParent 		:= B,
							sObjectName		:= '{F01}',		
							sDescription	:= '{Floor 01}',
							eDPADMode		:= E_BA_DPADMode.eInclude					
						);  
// Level 3 Gewerk Automationsschwerpunkt
// Level 3 Trade AutomationFocalPoint                                                                                       	
				ACE			: FB_BA_AutomationControl := (
								iParent 		:= F01,
								sObjectName		:= '{ACE}',
								sDescription	:= '{Automation Control}',			
								eDPADMode		:= E_BA_DPADMode.eInclude					
							);     
// Level 3 Gewerk Gebäudeautomation Allgemein   
// Level 3 Trade General                                                                                       	
				BAG			: FB_BA_BuildingAutomation := (
								iParent 		:= F01,
								sObjectName		:= '{BAG}',
								sDescription	:= '{Building Automation}',			
								eDPADMode		:= E_BA_DPADMode.eInclude					
							);  	 											   	 											

// Level 3 Gewerk Luftechnische Anlagen      
// Level 3 Trade ventilation system        
				ACS			: FB_BA_AirConditioning := (
								iParent 		:= F01,
								sObjectName		:= '{ACS}',
								sDescription	:= '{Air Conditioning}',  									
								eDPADMode		:= E_BA_DPADMode.eInclude					
							);  			                                                                        	
// Level 3 Gewerk Wärmeversorgungsanlagen  
// Level 3 Trade Heat supply systems, heat distribution  --> 	HD = heat distribution, HG = heat generation
				HTG			: FB_BA_Heating := (
								iParent 		:= F01,
								sObjectName		:= '{HTG}',
								sDescription	:= '{Heating}',        		
								eDPADMode		:= E_BA_DPADMode.eInclude			
							);     	    
// Level 3 Gewerk Raumautomation    
// Level 3 Trade room automation                                                                              	
				ROM			: FB_BA_RoomAutomation := (
								iParent			:= F01,
								sObjectName		:= '{ROM}',
								sDescription	:= '{Room automation}',        											
								eDPADMode		:= E_BA_DPADMode.eInclude
							); 

// SystemTime Settings								
	BACnetTime_TO_SysTime		: FB_BA_BACnetTime_TO_SysTime;	
	ExternalSysTime				: FB_BA_ExternalSysTime;
END_VAR


//	Level 1 Gebäude 	Building		
	B();
// Level 2 Stockwerk -->	O01 = Obergeschoss 01, U01 = Untergeschoss 01,  E00 = Ergeschoss 	floor ->	F01 = floor 01, B01 = basement 01,  GFL = Ground floor
		F01();
// Level 3 Gewerk Wärmeversorgungsanlagen	Heat supply systems	
			HTG(); 	
// Level 3 Gewerk Automation		Trade Automation			
			ACE(); 							
// Level 3 Gewerk Gebäudeautomation Allgemein		Trade BuildingAutomationGeneral			
			BAG(); 								
// Level 3 Gewerk Lufttechnische Anlagen		Trade ventilation system	
			ACS(); 								
// Level 3 Gewerk Raumautomation	Trade room automation 
			ROM(); 		
						
						
//	BACnetTime_TO_SysTime();	
	ExternalSysTime();

END_PROGRAM

// ---- Templates/POUs/Trade/AutomationControl/FB_BA_AutomationControl.TcPOU
{region '#Template'}
	{attribute 'Version' := '5.0.0.0'}
	{attribute 'Tags' := '"LCID": "1031", "Text": "Trade, Plant, General"'}
	{attribute 'Tags' := '"LCID": "1033", "Text": "Trade, Plant, General"'}
	{attribute 'Using' := '"Type": "Template", "URI": "Site"'}
	{attribute 'Description' := '"LCID": "1031", "Text": "Aufruf der Anlagen des Gewerks Allgemein"'}
	{attribute 'Description' := '"LCID": "1033", "Text": "Calling the plants of the trade general"'}
{endregion}
FUNCTION_BLOCK FB_BA_AutomationControl EXTENDS FB_BA_View
VAR_INPUT
END_VAR
VAR_INPUT CONSTANT
	Device				: FB_BA_Device;											 
	EvtGroups			: FB_BA_EvtGroupsAMEV2017;											 
	Cabinet				: FB_BA_ControlCabinet;				 
END_VAR

SUPER^(); // FB_BA_View
Device(); // FB_BA_Device
EvtGroups(); // FB_BA_EvtGroupsAMEV2017
Cabinet(); // FB_BA_ControlCabinet

METHOD FB_init : BOOL
VAR_INPUT
	bInitRetains : BOOL; // if TRUE, the retain variables are initialized (warm start / cold start)
	bInCopyCode : BOOL;  // if TRUE, the instance afterwards gets moved into the copy code (online change)
END_VAR
Device.iParent					:= THIS^;
Device.iLabel					:= LblPlt_Automation_control_equipment;	
Device.sObjectName				:= '{Idx=01}';  
Device.eDPADMode				:= E_BA_DPADMode.eInclude;		

EvtGroups.iParent				:= THIS^;	
EvtGroups.iLabel				:= LblPlt_EventGroups;
EvtGroups.sObjectName			:= '{Idx=01}';  
EvtGroups.eDPADMode				:= E_BA_DPADMode.eInclude;									

Cabinet.iParent					:= THIS^;	
Cabinet.iLabel					:= LblPlt_Control_cabinet;
Cabinet.sObjectName				:= '{Idx=01}';  
Cabinet.eDPADMode				:= E_BA_DPADMode.eInclude;
END_METHOD

END_FUNCTION_BLOCK

// ---- Templates/POUs/Trade/AutomationControl/Device/FB_BA_Device.TcPOU
{region '#Template'}
	{attribute 'Version' := '5.0.1.0'}
	{attribute 'Tags' := '"LCID": "1031", "Text": "Automatisierungssteuerung, Gerät, Einstellungen, Projekt, Parameter, Trend, Empfängerliste"'}
	{attribute 'Tags' := '"LCID": "1033", "Text": "Automation control, Device, Settings, Project, Parameter, Trend, Recipient list"'}
	{attribute 'Description' := '"LCID": "1031", "Text": "Basis Einstellungen der Steuerung"'}
	{attribute 'Description' := '"LCID": "1033", "Text": "Basic settings of the control"'}
{endregion}
	 
FUNCTION_BLOCK FB_BA_Device EXTENDS FB_BA_View
VAR_INPUT
END_VAR
VAR_INPUT CONSTANT
	Trend				: FB_BA_TrendLogging;	
	Project				: FB_BA_ProjectEx;
	Parameter			: FB_BA_Parameter;	
END_VAR
VAR_OUTPUT
END_VAR
VAR
	tonDlyStartPLC		: TON;	
END_VAR

SUPER^(); // FB_BA_View
tonDlyStartPLC(IN := TRUE, PT := T#2000ms); // TON
BA2_Param.bDlyStartPLC := tonDlyStartPLC.Q;
Parameter(); // FB_BA_Parameter
Trend(); // FB_BA_TrendLogging
// connect a UPS-monitoring FB at this input
Project(); // FB_BA_ProjectEx

METHOD FB_init : BOOL
VAR_INPUT
	bInitRetains : BOOL; // if TRUE, the retain variables are initialized (warm start / cold start)
	bInCopyCode : BOOL;  // if TRUE, the instance afterwards gets moved into the copy code (online change)
END_VAR
Project.iParent						:= THIS^;
Project.iLabel						:= LblComp_Project;
Project.sObjectName					:= '{Idx=11,Idx=99}';
Project.tPrsData_DefaultPeriod 		:= T#30M;
Project.tPrsData_ComissioningPeriod := T#10M;

Trend.iParent						:= THIS^;
Trend.iLabel						:= LblCtl_TrendLogging;
Trend.eDPADMode						:= E_BA_DPADMode.eInclude;
END_METHOD

END_FUNCTION_BLOCK

// ---- Templates/POUs/Universal/Control/Trend/FB_BA_TrendLogging.TcPOU
{region '#Template'}
	{attribute 'Version' := '5.0.1.0'}
	{attribute 'Tags' := '"LCID": "1031", "Text": "Universal, Control, Trend"'}
	{attribute 'Tags' := '"LCID": "1033", "Text": "Universal, Control, Trend"'}
	{attribute 'Using' := '"Type": "Template", "URI": "EC_ID"'}
	{attribute 'Using' := '"Type": "Template", "URI": "BA2_Param"'}
	{attribute 'Description' := '"LCID": "1031", "Text": "Trend"'}
	{attribute 'Description' := '"LCID": "1033", "Text": "Trend"'}
{endregion}			 
FUNCTION_BLOCK FB_BA_TrendLogging EXTENDS FB_BA_View
VAR_INPUT
END_VAR
VAR_OUTPUT
END_VAR
VAR_INPUT CONSTANT
	Trends						: ARRAY[1..TREND_COUNT] OF FB_BA_Trend;								
END_VAR
VAR
	i							: UDINT;
END_VAR
VAR CONSTANT
	TREND_COUNT						: UDINT := 30;
END_VAR

SUPER^();

FOR i := 1 TO TREND_COUNT DO
	Trends[i]();
END_FOR

METHOD FB_init : BOOL
VAR_INPUT
	bInitRetains : BOOL; // if TRUE, the retain variables are initialized (warm start / cold start)
	bInCopyCode : BOOL;  // if TRUE, the instance afterwards gets moved into the copy code (online change)
END_VAR 
VAR
END_VAR
FOR i := 1 TO TREND_COUNT DO
	Trends[i].iParent					:= THIS^;
	Trends[i].iLabel					:= LblFun_ObjectTrendLog;
	Trends[i].bEnable					:= BA2_Param.bTrend_DefLogEnable;
	Trends[i].stStartTime				:= BA2_Param.stTrend_DefStartTime;
	Trends[i].stStopTime				:= BA2_Param.stTrend_DefStopTime;	
	Trends[i].nLogInterval 				:= BA2_Param.nTrend_DefLogInterval;
	Trends[i].bStopOnFull				:= BA2_Param.bTrend_DefStopOnFull;
	Trends[i].nBufferSize 				:= BA2_Param.nTrend_BufferSize;
	Trends[i].eLoggingType				:= BA2_Param.eTrend_DefLoggingType;	
	Trends[i].nEventClassID				:= EC_ID.NC80;
	Trends[i].nNotificationThreshold	:= BA2_Param.nTrend_DefNotificationThreshold;
	Trends[i].aEventTransitionText[1]	:= txtEvent_Offnormal;
	Trends[i].aEventTransitionText[2]	:= txtEvent_None;
	Trends[i].aEventTransitionText[3]	:= txtEvent_Normal;
	Trends[i].bEventDetectionEnable		:= FALSE;
END_FOR
END_METHOD

END_FUNCTION_BLOCK

// ---- Templates/POUs/Trade/AutomationControl/Device/Project/FB_BA_ProjectEx.TcPOU
{region '#Template'}
	{attribute 'Version' := '5.0.0.0'}
	{attribute 'Tags' := '"LCID": "1031", "Text": "Automatisierungssteuerung, Gerät, Einstellungen, Projekt"'}
	{attribute 'Tags' := '"LCID": "1033", "Text": "Automation control, Device, Settings, Project"'}
	{attribute 'Description' := '"LCID": "1031", "Text": "Projektspezifische Informationen"'}
	{attribute 'Description' := '"LCID": "1033", "Text": "Project specific informations"'}
{endregion}
	 
FUNCTION_BLOCK FB_BA_ProjectEx EXTENDS FB_BA_Project
VAR_INPUT CONSTANT PERSISTENT
	{attribute 'parameterCategory' := 'Persistent Data'}
	tPrsData_DefaultPeriod : TIME := T#30M;
	{attribute 'parameterCategory' := 'Persistent Data'}
	tPrsData_ComissioningPeriod : TIME := T#10M;
END_VAR
VAR_INPUT CONSTANT
	{attribute 'parameterCategory' := 'Persistent Data'}
	bPrsData_ManualWriteData : BOOL;
END_VAR
VAR_INPUT
	bWrtPrsOnPowerFail		: BOOL;
END_VAR
VAR_OUTPUT
	nPrsDataWritten			: UINT;
END_VAR

SUPER^();

OnInitCycle();
PersistentData();

METHOD PROTECTED OnInitCycle
VAR
	_stVersion		: ST_LibVersion;
END_VAR
VAR CONSTANT
	FORMAT			: STRING		:= '%d.%d.%d.%d';
END_VAR
CASE (State) OF
	E_BA_ObjectState.eInstanceInit1:
		// Refresh runtime information:
		{IF defined (pou: F_GetVersion)}
			_stVersion := F_GetVersion();
			
			XBA_Globals.FormatStr2(
				pFormatString := ADR(FORMAT),
				arg1:=F_UINT(_stVersion.iMajor),
				arg2:=F_UINT(_stVersion.iMinor),
				arg3:=F_UINT(_stVersion.iBuild),
				arg4:=F_UINT(_stVersion.iRevision),
			
				pDstString := ADR(fbDiag.stVersion.Project),
				nDstSize := SIZEOF(fbDiag.stVersion.Project)
			);
		{END_IF}
		
END_CASE
END_METHOD

METHOD PROTECTED PersistentData
VAR_INST
	nOnlineChangeCnt		:	UDINT;
	iStep					:	INT;
	fbTon					:	TON;
	fbResetOnlineChange		:	TON;
	rtigManual				:	R_TRIG;
	trigUPS					:	R_TRIG;
	rFinishTrig				:	R_TRIG;
	WrtPersistDat			:	FB_BA_WrtPersistDat;
END_VAR
VAR CONSTANT
	DETECT_COMISSIONING_DURATION : TIME := T#60M;
END_VAR
IF	TwinCAT_SystemInfoVarList._AppInfo.OnlineChangeCnt <> nOnlineChangeCnt THEN
	nOnlineChangeCnt := TwinCAT_SystemInfoVarList._AppInfo.OnlineChangeCnt;
	fbResetOnlineChange(IN := FALSE);
	fbTon(IN := FALSE);
	iStep := 10;
END_IF

IF	tPrsData_DefaultPeriod < T#600S THEN
	tPrsData_DefaultPeriod	:= T#1800S;
END_IF

IF	tPrsData_ComissioningPeriod < T#30S THEN
	tPrsData_ComissioningPeriod	:= T#300S;
END_IF

CASE	iStep	OF
	0:
		fbTon(IN := NOT fbTon.Q,PT := tPrsData_DefaultPeriod);
	10:
		fbTon(IN := NOT fbTon.Q,PT := tPrsData_ComissioningPeriod);
		fbResetOnlineChange(IN := TRUE, PT := DETECT_COMISSIONING_DURATION);
		
		IF	fbResetOnlineChange.Q THEN
			iStep := 0;
			fbResetOnlineChange(IN := FALSE);
		END_IF
END_CASE
 
rtigManual(CLK := bPrsData_ManualWriteData);
bPrsData_ManualWriteData := FALSE;

trigUPS(CLK := bWrtPrsOnPowerFail);

// Write persistent data:
WrtPersistDat(bStt:=(fbTon.Q OR rtigManual.Q OR trigUPS.Q));
rFinishTrig(CLK:=(WrtPersistDat.bBusy AND NOT WrtPersistDat.bErr));

IF (rFinishTrig.Q) THEN
	nPrsDataWritten := (nPrsDataWritten+1);
END_IF
END_METHOD

END_FUNCTION_BLOCK

// ---- Templates/POUs/Trade/AutomationControl/Device/BACnetSettings/FB_BA_Parameter.TcPOU
{region '#Template'}
	{attribute 'Version' := '5.0.0.0'}
	{attribute 'Tags' := '"LCID": "1031", "Text": "Automatisierungssteuerung, Gerät, Einstellungen, Projekt, Parameter"'}
	{attribute 'Tags' := '"LCID": "1033", "Text": "Automation control, Device, Settings, Project, Parameter"'}
	{attribute 'Description' := '"LCID": "1031", "Text": "Basis Parameter"'}
	{attribute 'Description' := '"LCID": "1033", "Text": "Basic settings"'}
{endregion}

FUNCTION_BLOCK FB_BA_Parameter
VAR_INPUT
END_VAR
VAR_OUTPUT
END_VAR
VAR		
//		Recipient		: FB_BACnet_RcpList;	
END_VAR

// Recipient list to write (to all event classes):
// Recipient();

METHOD FB_init : BOOL
VAR_INPUT
	bInitRetains : BOOL; // if TRUE, the retain variables are initialized (warm start / cold start)
	bInCopyCode : BOOL;  // if TRUE, the instance afterwards gets moved into the copy code (online change)
END_VAR
VAR
	Parameters 				: FB_BA_Param;	
END_VAR
//Writeaccess on EventEnable Bits (Property 35.)
Parameters.SetDefWriteAccess(E_BA_Parameter.eEventEnable, E_BA_ROLE.eInternal);

//DefaultSeparator on each DPAD Level
Parameters.DPAD_ObjectName_DefSeparator:='-';
Parameters.DPAD_Description_DefSeparator:=' - ';

//Default structure of BACnetObjects in Systemmanager 
Parameters.BACnet_View_SubordinateAnnotationMode := Tc3_BACnetRev14.E_BACnet_AnnotationTitle.eObjectName;

//Set AckknowledgeRequiredFlags to AMEV 2017 Standard (Property 1.)
Parameters.AckFlags_Simple 		:= F_BA_EventTransition(bToOffNormal:= FALSE, bToFault:=FALSE, bToNormal:=FALSE);
Parameters.AckFlags_Standard	:= F_BA_EventTransition(bToOffNormal:= TRUE, bToFault:=FALSE, bToNormal:=FALSE);
Parameters.AckFlags_Extended 	:= F_BA_EventTransition(bToOffNormal:= TRUE, bToFault:=FALSE, bToNormal:=TRUE);

//Set EventEnable to AMEV 2017 Standard (Property 35.)
Parameters.EventEn_Simple 		:= F_BA_EventTransition(bToOffNormal:= TRUE, bToFault:=FALSE, bToNormal:=TRUE);
Parameters.EventEn_Standard		:= F_BA_EventTransition(bToOffNormal:= TRUE, bToFault:=FALSE, bToNormal:=TRUE);
Parameters.EventEn_Extended		:= F_BA_EventTransition(bToOffNormal:= TRUE, bToFault:=FALSE, bToNormal:=TRUE);

// Quittier- und Rücksetzmodus	// Acknowledge mode
// E_BA_AcknowledgeMode.eSingle	// Acknowledges only the next outstanding event transition by executing an acknowledgement.
// E_BA_AcknowledgeMode.eEntire	// Acknowledges all unacknowledged event transitions by executing a single acknowledgement.
Parameters.EvtMgmt_AckMode		:= E_BA_AcknowledgeMode.eSingle;
END_METHOD

END_FUNCTION_BLOCK

// ---- Templates/POUs/Trade/AutomationControl/EventClasses/FB_BA_EvtGroupsAMEV2017.TcPOU
{region '#Template'}
	{attribute 'Version' := '5.0.0.0'}
	{attribute 'Tags' := '"LCID": "1031", "Text": "General, Cabinet, Control cabinet, Event groups, Categories, Notification classes, Event classes"'}
	{attribute 'Tags' := '"LCID": "1033", "Text": "General, Cabinet, Control cabinet, Event groups, Categories, Notification classes, Event classes"'}
	{attribute 'Using' := '"Type": "Template", "URI": "EC_ID"'}
	{attribute 'Description' := '"LCID": "1031", "Text": "Ereignisgruppen, Kategorien"'}
	{attribute 'Description' := '"LCID": "1033", "Text": "Event groups, categories"'}
{endregion}
FUNCTION_BLOCK FB_BA_EvtGroupsAMEV2017 EXTENDS FB_BA_View
VAR_INPUT CONSTANT
	LifeSafety						: FB_BA_EvtCategory;
	SafetyMsg						: FB_BA_EvtCategory;
	AlarmMsg						: FB_BA_EvtCategory;
	FaultMsg						: FB_BA_EvtCategory;
	MaintenanceMsg01				: FB_BA_EvtCategory;
	MaintenanceMsg02				: FB_BA_EvtCategory;
	SystemMsg						: FB_BA_EvtCategory;
	ManualOp						: FB_BA_EvtCategory;
	OtherMsg						: FB_BA_EvtCategory;
END_VAR

SUPER^(); // FB_BA_View
LifeSafety(); // FB_BA_EvtCategory
SafetyMsg(); // FB_BA_EvtCategory
AlarmMsg(); // FB_BA_EvtCategory
FaultMsg(); // FB_BA_EvtCategory
MaintenanceMsg01(); // FB_BA_EvtCategory
MaintenanceMsg02(); // FB_BA_EvtCategory
SystemMsg(); // FB_BA_EvtCategory
ManualOp(); // FB_BA_EvtCategory
OtherMsg(); // FB_BA_EvtCategory

METHOD FB_init : BOOL
VAR_INPUT
	bInitRetains : BOOL; // if TRUE, the retain variables are initialized (warm start / cold start)
	bInCopyCode : BOOL;  // if TRUE, the instance afterwards gets moved into the copy code (online change)
END_VAR
//===================================================================
// Ereigniskategorie - Gefahr für Leben // Event category - Danger to life
// Brandalarm, Überfall // Fire alarm, robbery
LifeSafety.iParent							:= THIS^;
LifeSafety.iLabel							:= LblCtl_EvtCategoryLifeSafty;
LifeSafety.eDPADMode						:= E_BA_DPADMode.eInclude;																						
LifeSafety.EC.nInstanceID					:= EC_ID.NC10;
LifeSafety.EC.iLabel						:= LblFun_ObjectNotificationClass;
LifeSafety.EC.sObjectName					:='{Idx=10}';
LifeSafety.EC.eAlarmMode					:= E_BA_AlarmMode.eExtended;
LifeSafety.EC.eEventType					:= E_BA_EventType.eAlarm;
LifeSafety.EC.aPriority[1]					:= 10;
LifeSafety.EC.aPriority[2]					:= 11;
LifeSafety.EC.aPriority[3]					:= 12;
//===================================================================		
// Ereigniskategorie - Gefahrenmeldung, Sicherheitsmeldung // Event category - hazard alert, safety message
// Einbruch, unberechtigter Zutritt // Burglary, unauthorised entry
SafetyMsg.iParent							:= THIS^;
SafetyMsg.iLabel							:= LblCtl_EvtCategorySaftyMessage;
SafetyMsg.eDPADMode							:= E_BA_DPADMode.eInclude;																						
SafetyMsg.EC.nInstanceID					:= EC_ID.NC20;
SafetyMsg.EC.iLabel							:= LblFun_ObjectNotificationClass;
SafetyMsg.EC.sObjectName					:='{Idx=20}';
SafetyMsg.EC.eAlarmMode						:= E_BA_AlarmMode.eExtended;
SafetyMsg.EC.eEventType						:= E_BA_EventType.eAlarm;
SafetyMsg.EC.aPriority[1]					:= 40;
SafetyMsg.EC.aPriority[2]					:= 41;
SafetyMsg.EC.aPriority[3]					:= 42;
//===================================================================//
// Ereigniskategorie - Alarmeldung - Meldung signalisiert Anlagenausfall oder erfordert sofortigen Eingriff 
// Event category - Alarm message - Message signals system failure or requires immediate intervention 
// Sicherheitstemperaturbegrenzer (STB), Sicherheitsdruckbegrenzer (SDB), Übertemperatur der Warmwasserbereitung (WWB), Sicherheitsventile, Hauptpumpen, Keilriemenwächter, Frequenzumformer, Kälteanlagen, Spannungsausfall usw
// Safety temperature limiter, safety pressure limiter, excess temperature of water heating, safety valves, main pumps, V-belt monitors, frequency converters, refrigeration systems, voltage failure, etc.
AlarmMsg.iParent							:= THIS^;
AlarmMsg.iLabel								:= LblCtl_EvtCategoryAlarmMessage;
AlarmMsg.eDPADMode							:= E_BA_DPADMode.eInclude;																						
AlarmMsg.EC.nInstanceID						:= EC_ID.NC30;
AlarmMsg.EC.iLabel							:= LblFun_ObjectNotificationClass;
AlarmMsg.EC.sObjectName						:= '{Idx=30}'	;
AlarmMsg.EC.eAlarmMode						:= E_BA_AlarmMode.eExtended;
AlarmMsg.EC.eEventType						:= E_BA_EventType.eAlarm;
AlarmMsg.EC.aPriority[1]					:= 70;
AlarmMsg.EC.aPriority[2]					:= 71;
AlarmMsg.EC.aPriority[3]					:= 72;
//===================================================================
// Ereigniskategorie - Störungsmeldung - Meldung weist auf einen anormalen Betriebszustand hin
// Event category - malfunction message - message indicates abnormal operating condition
// Temperaturwächter (TW), Druckwächter (DW), Temperaturüberwachung von Wärmetauscher (WT) und WWB, Motorschutz, Aufzug-Sammelstörmeldung, Netzdrücke usw.
// Temperature monitor, pressure monitor, temperature monitoring of heat exchanger and water heating, motor protection, lift collective fault signal, mains pressures, etc.
FaultMsg.iParent							:= THIS^;
FaultMsg.iLabel								:= LblCtl_EvtCategoryFaultMessage;
FaultMsg.eDPADMode							:= E_BA_DPADMode.eInclude;																						
FaultMsg.EC.nInstanceID						:= EC_ID.NC40;
FaultMsg.EC.iLabel							:= LblFun_ObjectNotificationClass;
FaultMsg.EC.sObjectName						:= '{Idx=40}'	;
FaultMsg.EC.eAlarmMode						:= E_BA_AlarmMode.eStandard;
FaultMsg.EC.eEventType						:= E_BA_EventType.eDisturb;
FaultMsg.EC.aPriority[1]					:= 100;
FaultMsg.EC.aPriority[2]					:= 101;
FaultMsg.EC.aPriority[3]					:= 102;
//===================================================================
// Ereigniskategorie - Wartungsmeldung, Hinweis auf Wartungsaktivität o.ä.
// Event category - Maintenance message Maintenance message, indication of maintenance activity or similar.
// Betriebsstunden, Behälterstand, Reparaturschalter usw.
// Operating hours, tank level, repair switch, etc.
MaintenanceMsg01.iParent					:= THIS^;
MaintenanceMsg01.iLabel						:= LblCtl_EvtCategoryMaintenanceMessage;
MaintenanceMsg01.eDPADMode					:= E_BA_DPADMode.eInclude;																						
MaintenanceMsg01.EC.nInstanceID				:= EC_ID.NC50;
MaintenanceMsg01.EC.iLabel					:= LblFun_ObjectNotificationClass;
MaintenanceMsg01.EC.sObjectName				:= '{Idx=50}'	;
MaintenanceMsg01.EC.eAlarmMode				:= E_BA_AlarmMode.eStandard;
MaintenanceMsg01.EC.eEventType				:= E_BA_EventType.eMaintenance;
MaintenanceMsg01.EC.aPriority[1]			:= 130;
MaintenanceMsg01.EC.aPriority[2]			:= 131;
MaintenanceMsg01.EC.aPriority[3]			:= 132;
// Filterende erreicht, Filter verschmutzt usw.
// Filter end reached, filter dirty, etc.
MaintenanceMsg02.iParent					:= THIS^;
MaintenanceMsg02.iLabel						:= LblCtl_EvtCategoryMaintenanceMessage;
MaintenanceMsg02.eDPADMode					:= E_BA_DPADMode.eInclude;																						
MaintenanceMsg02.EC.nInstanceID				:= EC_ID.NC51;
MaintenanceMsg02.EC.iLabel					:= LblFun_ObjectNotificationClass;
MaintenanceMsg02.EC.sObjectName				:= '{Idx=51}'	;
MaintenanceMsg02.EC.eAlarmMode				:= E_BA_AlarmMode.eStandard;
MaintenanceMsg02.EC.eEventType				:= E_BA_EventType.eMaintenance;
MaintenanceMsg02.EC.aPriority[1]			:= 135;
MaintenanceMsg02.EC.aPriority[2]			:= 136;
MaintenanceMsg02.EC.aPriority[3]			:= 137;
//===================================================================
//===================================================================
// Ereigniskategorie - Systemmeldung, Störungsmeldung aus GA-System
// Event category - System message, System message, Fault message from building automation system
// Gerätestörung, Batteriemeldung, Kommunikationsunterbrechung usw.
// Unit malfunction, battery message, communication interruption, etc.
SystemMsg.iParent							:= THIS^;
SystemMsg.iLabel							:= LblCtl_EvtCategorySystem;
SystemMsg.eDPADMode							:= E_BA_DPADMode.eInclude;																						
SystemMsg.EC.nInstanceID					:= EC_ID.NC60;
SystemMsg.EC.iLabel							:= LblFun_ObjectNotificationClass;
SystemMsg.EC.sObjectName					:='{Idx=60}';
SystemMsg.EC.eAlarmMode						:= E_BA_AlarmMode.eSimple;
SystemMsg.EC.eEventType						:= E_BA_EventType.eNotification;
SystemMsg.EC.aPriority[1]					:= 180;
SystemMsg.EC.aPriority[2]					:= 181;
SystemMsg.EC.aPriority[3]					:= 182;
//===================================================================//
//	Ereigniskategorie - Manual operation, Handeingriff
ManualOp.iParent							:= THIS^;
ManualOp.iLabel								:= LblCtl_EvtCategoryManualOperation;
ManualOp.eDPADMode							:= E_BA_DPADMode.eInclude;																						
ManualOp.EC.nInstanceID						:= EC_ID.NC70;
ManualOp.EC.iLabel							:= LblFun_ObjectNotificationClass;
ManualOp.EC.sObjectName						:='{Idx=70}';
ManualOp.EC.eAlarmMode						:= E_BA_AlarmMode.eSimple;
ManualOp.EC.eEventType						:= E_BA_EventType.eOther;
ManualOp.EC.aPriority[1]					:= 220;
ManualOp.EC.aPriority[2]					:= 220;
ManualOp.EC.aPriority[3]					:= 220;
//===================================================================//
// Ereigniskategorie - Freibleibend, Sonstige Meldungen
// Event category - Other message, Not binding, Other messages
// Betriebszustandswechsel, Betriebsarten, Trendspeicher voll usw.
// Operating status change, operating modes, trend memory full, etc.
OtherMsg.iParent							:= THIS^;
OtherMsg.iLabel								:= LblCtl_EvtCategoryOther;
OtherMsg.eDPADMode							:= E_BA_DPADMode.eInclude;																						
OtherMsg.EC.nInstanceID						:= EC_ID.NC80;
OtherMsg.EC.iLabel							:= LblFun_ObjectNotificationClass;
OtherMsg.EC.sObjectName						:='{Idx=80}';
OtherMsg.EC.eAlarmMode						:= E_BA_AlarmMode.eSimple;
OtherMsg.EC.eEventType						:= E_BA_EventType.eOther;
OtherMsg.EC.aPriority[1]					:= 230;
OtherMsg.EC.aPriority[2]					:= 231;
OtherMsg.EC.aPriority[3]					:= 232;
END_METHOD

END_FUNCTION_BLOCK

// ---- Templates/POUs/Universal/Control/EventClasses/FB_BA_EvtCategory.TcPOU
{region '#Template'}
	{attribute 'Version' := '5.0.0.0'}
	{attribute 'Tags' := '"LCID": "1031", "Text": "Universal, Control, Event class, Notification"'}
	{attribute 'Tags' := '"LCID": "1033", "Text": "Universal, Control, Event class, Notification"'}
	{attribute 'Using' := '"Type": "Template", "URI": "EC_ID"'}
	{attribute 'Description' := '"LCID": "1031", "Text": "Ereignisklasse"'}
	{attribute 'Description' := '"LCID": "1033", "Text": "Event class"'}
{endregion}
FUNCTION_BLOCK FB_BA_EvtCategory EXTENDS FB_BA_View
VAR_INPUT CONSTANT
		EC				: FB_BA_EC;  
END_VAR

SUPER^(); // FB_BA_View
EC(); // FB_BA_EC

METHOD FB_init : BOOL
VAR_INPUT
	bInitRetains : BOOL; // if TRUE, the retain variables are initialized (warm start / cold start)
	bInCopyCode : BOOL;  // if TRUE, the instance afterwards gets moved into the copy code (online change)
END_VAR
EC.iParent					:= THIS^;
EC.iLabel					:= LblCtl_EvtClass;   
EC.nInstanceID				:= EC_ID.NC10;
EC.eEventType				:= E_BA_EventType.eAlarm;
EC.aPriority[1]				:= 16;
EC.aPriority[2]				:= 17;
EC.aPriority[3]				:= 18;
END_METHOD

END_FUNCTION_BLOCK

// ---- Templates/POUs/Trade/AutomationControl/ControlCabinet/FB_BA_ControlCabinet.TcPOU
{region '#Template'}
	{attribute 'Version' := '5.0.0.0'}
	{attribute 'Tags' := '"LCID": "1031", "Text": "General, Cabinet, Control cabinet"'}
	{attribute 'Tags' := '"LCID": "1033", "Text": "General, Cabinet, Control cabinet"'}
	{attribute 'Using' := '"Type": "Template", "URI": "EC_ID"'}
	{attribute 'Description' := '"LCID": "1031", "Text": "Schaltschrank Ereignisse"'}
	{attribute 'Description' := '"LCID": "1033", "Text": "Control cabinet events"'}
{endregion}
FUNCTION_BLOCK FB_BA_ControlCabinet EXTENDS FB_BA_ControlCabinetBasic
VAR_INPUT CONSTANT
	Fuse01					: FB_BA_SensorBinary_Raw;		
	Fuse02					: FB_BA_SensorBinary_Raw;	
	Fuse03					: FB_BA_SensorBinary_Raw;	
END_VAR

SUPER^(); // FB_BA_ControlCabinetBasic
Fuse01(); // FB_BA_SensorBinary_Raw
Fuse02(); // FB_BA_SensorBinary_Raw
Fuse03(); // FB_BA_SensorBinary_Raw

METHOD FB_init : BOOL
VAR_INPUT
	bInitRetains : BOOL; // if TRUE, the retain variables are initialized (warm start / cold start)
	bInCopyCode : BOOL;  // if TRUE, the instance afterwards gets moved into the copy code (online change)
END_VAR
Fuse01.iParent								:= THIS^;
Fuse01.iLabel								:= LblCtl_Fuse;
Fuse01.sObjectName							:='{Idx=10}';	
Fuse01.eDPADMode							:= E_BA_DPADMode.eInclude;	
Fuse01.Input.iLabel							:= LblFun_Fault;																																									
Fuse01.Input.ePolarity						:= E_BA_Polarity.eReverse;
Fuse01.Input.sActiveText 					:= txtEvent_Triggered;
Fuse01.Input.sInactiveText 					:= txtEvent_Normal;
Fuse01.Input.nEventClassID					:= EC_ID.NC30;
Fuse01.Input.aEventTransitionText[1]		:= txtEvent_Triggered;
Fuse01.Input.aEventTransitionText[2]		:= txtEvent_Error;
Fuse01.Input.aEventTransitionText[3]		:= txtEvent_Normal;
Fuse01.Input.bEventDetectionEnable			:= TRUE;

Fuse01.Input.eEnPlantLock					:= E_BA_LockPriority.eNoLock;	
								 
Fuse02.iParent								:= THIS^;		
Fuse02.iLabel								:= LblCtl_Fuse;	
Fuse02.sObjectName							:='{Idx=20}';	
Fuse02.eDPADMode							:= E_BA_DPADMode.eInclude;	
Fuse02.Input.iLabel							:= LblFun_Fault;																				
Fuse02.Input.ePolarity						:= E_BA_Polarity.eReverse;
Fuse02.Input.sActiveText 					:= txtEvent_Triggered;
Fuse02.Input.sInactiveText 					:= txtEvent_Normal;
Fuse02.Input.nEventClassID					:= EC_ID.NC30;
Fuse02.Input.aEventTransitionText[1]		:= txtEvent_Triggered;
Fuse02.Input.aEventTransitionText[2]		:= txtEvent_Error;
Fuse02.Input.aEventTransitionText[3]		:= txtEvent_Normal;
Fuse02.Input.bEventDetectionEnable			:= TRUE;

Fuse02.Input.eEnPlantLock					:= E_BA_LockPriority.eNoLock;	
										 
Fuse03.iParent								:= THIS^;		
Fuse03.iLabel								:= LblCtl_Fuse;	
Fuse03.sObjectName							:='{Idx=30}';	
Fuse03.eDPADMode							:= E_BA_DPADMode.eInclude;				
Fuse03.Input.iLabel							:= LblFun_Fault;																				
Fuse03.Input.ePolarity						:= E_BA_Polarity.eReverse;
Fuse03.Input.sActiveText 					:= txtEvent_Triggered;
Fuse03.Input.sInactiveText 					:= txtEvent_Normal;
Fuse03.Input.nEventClassID					:= EC_ID.NC30;
Fuse03.Input.aEventTransitionText[1]		:= txtEvent_Triggered;
Fuse03.Input.aEventTransitionText[2]		:= txtEvent_Error;
Fuse03.Input.aEventTransitionText[3]		:= txtEvent_Normal;
Fuse03.Input.bEventDetectionEnable			:= TRUE;

Fuse03.Input.eEnPlantLock					:= E_BA_LockPriority.eNoLock;
END_METHOD

END_FUNCTION_BLOCK

// ---- Templates/POUs/Trade/AutomationControl/ControlCabinet/FB_BA_ControlCabinetBasic.TcPOU
{region '#Template'}
	{attribute 'Version' := '5.0.0.0'}
	{attribute 'Tags' := '"LCID": "1031", "Text": "General, Cabinet, Control cabinet, Acknowledgement"'}
	{attribute 'Tags' := '"LCID": "1033", "Text": "General, Cabinet, Control cabinet, Acknowledgement"'}
	{attribute 'Using' := '"Type": "Template", "URI": "BA2_Param"'}
	{attribute 'Using' := '"Type": "Template", "URI": "EC_ID"'}
	{attribute 'Description' := '"LCID": "1031", "Text": "Schaltschrank Quittierung"'}
	{attribute 'Description' := '"LCID": "1033", "Text": "Control cabinet acknowledgement"'}
{endregion}
FUNCTION_BLOCK FB_BA_ControlCabinetBasic EXTENDS FB_BA_View
VAR_INPUT CONSTANT
	LampFault				: FB_BA_ActuatorCmd;		
	AckButton				: FB_BA_CombinationBI_BV;													
	RstHw					: FB_BA_ActuatorCmd;	
	EventObserver			: FB_BA_EventObserver;													
END_VAR
VAR				
	bHasEvents				: BOOL;
	bHasUnackEvent			: BOOL;
	tpResetHw				: TP;	
	bTrigRstSwi				: BOOL;
	bTrigRstButton			: BOOL;	
	Blink					: FB_BA_Blink;
END_VAR
VAR // added by the converter: edge detectors and wires of the graphical bodies
    _s1, _s2 : ST_BA_Binary;
END_VAR

SUPER^(); // FB_BA_View
AckButton(); // FB_BA_CombinationBI_BV
bTrigRstSwi := AckButton.bTrigBI_PrVal;
bTrigRstButton := AckButton.bTrigBV_PrVal;
EventObserver(bAck := bTrigRstSwi OR bTrigRstButton); // FB_BA_EventObserver
bHasEvents := EventObserver.bHasEvents;
bHasUnackEvent := EventObserver.bHasUnackEvents;
// compose _s1 : ST_BA_Binary
_s1.bEnPgm := bHasEvents;
_s1.bValPgm := SEL(bHasUnackEvent, TRUE, BA2_Param.bBlink);
LampFault(stCmd := _s1); // FB_BA_ActuatorCmd
Blink(bEn := TRUE, nTiOn := 800, nTiOff := 800); // FB_BA_Blink
BA2_Param.bBlink := Blink.bQ;
tpResetHw(IN := bTrigRstSwi OR bTrigRstButton, PT := T#2s); // TP
// compose _s2 : ST_BA_Binary
_s2.bEnPgm := TRUE;
_s2.bValPgm := tpResetHw.Q;
RstHw(stCmd := _s2); // FB_BA_ActuatorCmd

METHOD FB_init : BOOL
VAR_INPUT
	bInitRetains : BOOL; // if TRUE, the retain variables are initialized (warm start / cold start)
	bInCopyCode : BOOL;  // if TRUE, the instance afterwards gets moved into the copy code (online change)
END_VAR
LampFault.iParent							:= THIS^;
LampFault.iLabel							:= LblCtl_EventIndicationLamp;
LampFault.eDPADMode							:= E_BA_DPADMode.eInclude;	
LampFault.Cmd.iLabel						:= LblFun_SwitchingCommand;		
LampFault.Cmd.ePolarity						:= E_BA_Polarity.eNormal;
LampFault.Cmd.sActiveText 					:= txtEvent_On;
LampFault.Cmd.sInactiveText 				:= txtEvent_Off;
LampFault.Cmd.nEventClassID					:= EC_ID.NC40;
LampFault.Cmd.aEventTransitionText[1]		:= txtEvent_Disturb;
LampFault.Cmd.aEventTransitionText[2]		:= txtEvent_None;
LampFault.Cmd.aEventTransitionText[3]		:= txtEvent_Normal;
LampFault.Cmd.bEventDetectionEnable			:= FALSE;
LampFault.Cmd.eEnPlantLock					:= E_BA_LockPriority.eNoLock;	

AckButton.iParent							:= THIS^;
AckButton.iLabel							:= LblCtl_Acknowledge;				
AckButton.eDPADMode							:= E_BA_DPADMode.eInclude;
AckButton.Input.iLabel						:= LblCtl_ButtonLocalAcknowledgement;																										
AckButton.Input.ePolarity					:= E_BA_Polarity.eNormal;
AckButton.Input.bEventDetectionEnable		:= FALSE;
AckButton.Value.eToggleMode 				:= E_BA_ToggleMode.ePushButton;					

RstHw.iParent								:= THIS^;
RstHw.iLabel								:= LblCtl_AcknowledgeCommand;		
RstHw.eDPADMode								:= E_BA_DPADMode.eInclude;	
RstHw.Cmd.iLabel							:= LblFun_SwitchingCommand;		
RstHw.Cmd.ePolarity							:= E_BA_Polarity.eNormal;
RstHw.Cmd.sActiveText 						:= txtEvent_On;
RstHw.Cmd.sInactiveText 					:= txtEvent_Off;
RstHw.Cmd.nEventClassID						:= EC_ID.NC40;
RstHw.Cmd.aEventTransitionText[1]			:= txtEvent_Disturb;
RstHw.Cmd.aEventTransitionText[2]			:= txtEvent_None;
RstHw.Cmd.aEventTransitionText[3]			:= txtEvent_Normal;
RstHw.Cmd.bEventDetectionEnable				:= FALSE;
RstHw.Cmd.eEnPlantLock						:= E_BA_LockPriority.eNoLock;	

EventObserver.Parent						:= XBA_Globals.Top;
END_METHOD

END_FUNCTION_BLOCK

// ---- Templates/POUs/Universal/Aggregat/Binary/FB_BA_ActuatorCmd.TcPOU
{region '#Template'}
	{attribute 'Version' := '5.0.0.0'}
	{attribute 'Tags' := '"LCID": "1031", "Text": "Universal, Analog, Aggregate"'}
	{attribute 'Tags' := '"LCID": "1033", "Text": "Universal, Analog, Aggregate"'}
	{attribute 'Using' := '"Type": "Template", "URI": "EC_ID"'}
	{attribute 'Using' := '"Type": "Template", "URI": "BA2_Param"'}
	{attribute 'Description' := '"LCID": "1031", "Text": "Aktor binär"'}
	{attribute 'Description' := '"LCID": "1033", "Text": "Actuator binary"'}
{endregion}
FUNCTION_BLOCK FB_BA_ActuatorCmd EXTENDS FB_BA_View
VAR_INPUT
	stCmd						: ST_BA_Binary;	
END_VAR
VAR_OUTPUT
	bCmd						: BOOL;
	bDst						: BOOL;
	eActivePrio					: E_BA_Priority;
END_VAR
VAR_INPUT CONSTANT
	Cmd							: FB_BA_BO_Raw;		
	PlantLock					: FB_BA_PlantLock;								
END_VAR
VAR
	bPrioSfty					: BOOL;
	bPrioCrit					: BOOL;	
END_VAR
VAR // added by the converter: edge detectors and wires of the graphical bodies
    _w1 : ANY;
END_VAR

SUPER^(); // FB_BA_View
PlantLock(); // FB_BA_PlantLock
bPrioSfty := PlantLock.bPrioHigh OR PlantLock.bPrioLocalHigh;
bPrioCrit := PlantLock.bPrioMedium OR PlantLock.bPrioLocalMedium;
bDst := bPrioSfty OR bPrioCrit;
Cmd(
    bEnSfty := stCmd.bEnSfty OR bPrioSfty,
    bValSfty := SEL(bPrioSfty, stCmd.bValSfty, FALSE),
    bEnCrit := stCmd.bEnCrit OR bPrioCrit,
    bValCrit := _w1,
    bEnPgm := stCmd.bEnPgm,
    bValPgm := stCmd.bValPgm); // FB_BA_BO_Raw
_w1 := SEL(bPrioCrit, stCmd.bValCrit, FALSE);
bCmd := Cmd.bPresentValue;
eActivePrio := Cmd.eActivePrio;

METHOD FB_init : BOOL
VAR_INPUT
	bInitRetains : BOOL; // if TRUE, the retain variables are initialized (warm start / cold start)
	bInCopyCode : BOOL;  // if TRUE, the instance afterwards gets moved into the copy code (online change)
END_VAR
PlantLock.Parent					:= THIS^;		

Cmd.iParent							:= THIS^;
Cmd.iLabel							:= LblFun_SwitchingCommand;  
Cmd.ePolarity						:= E_BA_Polarity.eNormal;
Cmd.sActiveText 					:= txtEvent_On;
Cmd.sInactiveText 					:= txtEvent_Off;
Cmd.bEnManualRm						:= FALSE;	//	Priority  8	
Cmd.bValManualRm					:= FALSE;	//	Priority  8
Cmd.nEventClassID					:= EC_ID.NC40;
Cmd.stTimeDelay.nToNormal			:= BA2_Param.nDefTimeDelay_ToNormal;
Cmd.stTimeDelay.nToAbnormal			:= BA2_Param.nDefTimeDelay_ToAbnormal;
Cmd.aEventTransitionText[1]			:= txtEvent_Disturb;
Cmd.aEventTransitionText[2]			:= txtEvent_None;
Cmd.aEventTransitionText[3]			:= txtEvent_Normal;
Cmd.bEventDetectionEnable			:= FALSE;
Cmd.eEnPlantLock					:= E_BA_LockPriority.eNoLock;
END_METHOD

END_FUNCTION_BLOCK

// ---- Templates/POUs/Universal/Sensor/FB_BA_CombinationBI_BV.TcPOU
{region '#Template'}
	{attribute 'Version' := '5.0.0.0'}
	{attribute 'Tags' := '"LCID": "1031", "Text": "Universal, Sensor, BI, BV"'}
	{attribute 'Tags' := '"LCID": "1033", "Text": "Universal, Sensor, BI, BV"'}
	{attribute 'Using' := '"Type": "Template", "URI": "EC_ID"'}
	{attribute 'Using' := '"Type": "Template", "URI": "BA2_Param"'}
	{attribute 'Description' := '"LCID": "1031", "Text": "Kombination aus BV BI"'}
	{attribute 'Description' := '"LCID": "1033", "Text": "Combination of BV BI"'}
{endregion}	 
FUNCTION_BLOCK FB_BA_CombinationBI_BV EXTENDS FB_BA_View
VAR_INPUT
END_VAR
VAR_INPUT CONSTANT
	Input				: FB_BA_BI_Raw;	
	Value				: FB_BA_BV_Op;									
END_VAR
VAR_OUTPUT
	bBI_PrVal			: BOOL;
	bTrigBI_PrVal		: BOOL;	
	bBV_PrVal			: BOOL;
	bTrigBV_PrVal		: BOOL;		
END_VAR
VAR
	TrigInput			: FB_BA_RFTrig;
	TrigValue			: FB_BA_RFTrig;
END_VAR

TrigInput(bValue := Input.bPresentValue); // FB_BA_RFTrig
TrigValue(bValue := Value.bPresentValue); // FB_BA_RFTrig
bTrigBI_PrVal := TrigInput.Qr;
bTrigBV_PrVal := TrigValue.Qr;
SUPER^(); // FB_BA_View
Input(); // FB_BA_BI_Raw
bBI_PrVal := Input.bPresentValue;
Value(); // FB_BA_BV_Op
bBV_PrVal := Value.bPresentValue;

METHOD FB_init : BOOL
VAR_INPUT
	bInitRetains : BOOL; // if TRUE, the retain variables are initialized (warm start / cold start)
	bInCopyCode : BOOL;  // if TRUE, the instance afterwards gets moved into the copy code (online change)
END_VAR
Input.iParent						:= THIS^;
Input.iLabel						:= LblFun_Button; 
Input.ePolarity						:= E_BA_Polarity.eReverse;
Input.sActiveText 					:= txtEvent_On;
Input.sInactiveText 				:= txtEvent_Off;
Input.nEventClassID					:= EC_ID.NC80;
Input.stTimeDelay.nToNormal			:= BA2_Param.nDefTimeDelay_ToNormal;
Input.stTimeDelay.nToAbnormal		:= BA2_Param.nDefTimeDelay_ToAbnormal;
Input.bAlarmValue					:= TRUE;
Input.aEventTransitionText[1]		:= txtEvent_Off;
Input.aEventTransitionText[2]		:= txtEvent_None;
Input.aEventTransitionText[3]		:= txtEvent_On;
Input.bEventDetectionEnable			:= FALSE;
Input.eEnPlantLock					:= E_BA_LockPriority.eNoLock;	

Value.iParent						:= THIS^;		
Value.iLabel						:= LblFun_Button; 
Value.sActiveText					:= txtEvent_On;
Value.sInactiveText					:= txtEvent_Off;
Value.bValueRm						:= FALSE;
Value.eToggleMode 					:= E_BA_ToggleMode.eSwitch;
END_METHOD

END_FUNCTION_BLOCK

// ---- Templates/POUs/Universal/Sensor/FB_BA_SensorBinary_Raw.TcPOU
{region '#Template'}
	{attribute 'Version' := '5.0.0.0'}
	{attribute 'Tags' := '"LCID": "1031", "Text": "Universal, Sensor, BI"'}
	{attribute 'Tags' := '"LCID": "1033", "Text": "Universal, Sensor, BI"'}
	{attribute 'Using' := '"Type": "Template", "URI": "EC_ID"'}
	{attribute 'Using' := '"Type": "Template", "URI": "BA2_Param"'}
	{attribute 'Description' := '"LCID": "1031", "Text": "BI mit IO"'}
	{attribute 'Description' := '"LCID": "1033", "Text": "BI with IO"'}
{endregion}		 
FUNCTION_BLOCK FB_BA_SensorBinary_Raw EXTENDS FB_BA_View
VAR_INPUT
END_VAR
VAR_INPUT CONSTANT
	Input					: FB_BA_BI_Raw;		
END_VAR
VAR_OUTPUT
	bPresentValue			: BOOL;	
END_VAR
VAR
END_VAR

SUPER^(); // FB_BA_View
Input(); // FB_BA_BI_Raw
bPresentValue := Input.bPresentValue;

METHOD FB_init : BOOL
VAR_INPUT
	bInitRetains : BOOL; // if TRUE, the retain variables are initialized (warm start / cold start)
	bInCopyCode : BOOL;  // if TRUE, the instance afterwards gets moved into the copy code (online change)
END_VAR
Input.iParent						:= THIS^;
Input.iLabel						:= LblFun_Fault;
Input.ePolarity						:= E_BA_Polarity.eReverse;
Input.sActiveText 					:= txtEvent_Triggered;
Input.sInactiveText 				:= txtEvent_Normal;
Input.nEventClassID					:= EC_ID.NC30;
Input.stTimeDelay.nToNormal			:= BA2_Param.nDefTimeDelay_ToNormal;
Input.stTimeDelay.nToAbnormal		:= BA2_Param.nDefTimeDelay_ToAbnormal;
Input.bAlarmValue					:= TRUE;
Input.aEventTransitionText[1]		:= txtEvent_Triggered;
Input.aEventTransitionText[2]		:= txtEvent_Error;
Input.aEventTransitionText[3]		:= txtEvent_Normal;
Input.bEventDetectionEnable			:= TRUE;
Input.eEnPlantLock					:= E_BA_LockPriority.eNoLock;
END_METHOD

END_FUNCTION_BLOCK

// ---- Templates/POUs/Trade/BuildingAutomation/FB_BA_BuildingAutomation.TcPOU
                                                                                                                                                                                                                                                {region '#Template'}
	{attribute 'Version' := '5.1.0.0'}
	{attribute 'Tags' := '"LCID": "1031", "Text": "Gewerk, Gebäudeautomation"'}
	{attribute 'Tags' := '"LCID": "1033", "Text": "Trade, Building automation"'}
	{attribute 'Using' := '"Type": "Template", "URI": "Site"'}
	{attribute 'Description' := '"LCID": "1031", "Text": "Aufruf der Anlagen des Gewerks Gebäudeautomation"'}
	{attribute 'Description' := '"LCID": "1033", "Text": "Calling the plants of the trade building automation"'}
{endregion}	 
	 
FUNCTION_BLOCK FB_BA_BuildingAutomation EXTENDS FB_BA_View
VAR_INPUT
END_VAR
VAR_INPUT CONSTANT
	BuildingGlobal		: FB_BA_EventsAndSettings;
	
	Weatherstation		: FB_BA_WeatherStation_Draft;			

	AdsComServer		: FB_BA_AdsComServer;	
//	AdsComClient		: FB_BA_AdsComClient;	
END_VAR

SUPER^(); // FB_BA_View
BuildingGlobal(fTWth := Site.stWeatherStation.fOutsideTemperature); // FB_BA_EventsAndSettings
Weatherstation(); // FB_BA_WeatherStation_Draft
AdsComServer(); // FB_BA_AdsComServer

METHOD FB_init : BOOL
VAR_INPUT
	bInitRetains : BOOL; // if TRUE, the retain variables are initialized (warm start / cold start)
	bInCopyCode : BOOL;  // if TRUE, the instance afterwards gets moved into the copy code (online change)
END_VAR
BuildingGlobal.iParent			:= THIS^;	
BuildingGlobal.iLabel			:= LblPlt_Global_Building_Data;
BuildingGlobal.sObjectName		:= '{Idx=01}';
BuildingGlobal.eDPADMode		:= E_BA_DPADMode.eInclude;
				 
Weatherstation.iParent			:= THIS^;
Weatherstation.iLabel			:= LblPlt_Weather_station;
Weatherstation.sObjectName		:= '{Idx=01}';
Weatherstation.eDPADMode		:= E_BA_DPADMode.eInclude;

// AdsComClient.iParent			:= THIS^;	
// AdsComClient.iLabel          := LblPlt_Global_Building_Data;
// AdsComClient.sObjectName		:= '{Idx=02}';
// AdsComClient.eDPADMode		:= E_BA_DPADMode.eInclude;
END_METHOD

END_FUNCTION_BLOCK

// ---- Templates/POUs/Trade/BuildingAutomation/GlobalEventsAndSettings/FB_BA_EventsAndSettings.TcPOU
{region '#Template'}
	{attribute 'Version' := '5.0.1.0'}
	{attribute 'Tags' := '"LCID": "1031", "Text": "Gebäudeautomation, Einstellungen, Parameter"'}
	{attribute 'Tags' := '"LCID": "1033", "Text": "Building automation, Settings, Parameters"'}
	{attribute 'Using' := '"Type": "Template", "URI": "Site"'}		 
	{attribute 'Description' := '"LCID": "1031", "Text": "Basis Parameter für die Templates"'}
	{attribute 'Description' := '"LCID": "1033", "Text": "Basic parameters for the templates"'}
{endregion}
FUNCTION_BLOCK FB_BA_EventsAndSettings EXTENDS FB_BA_View
VAR_INPUT
	fTWth					: REAL;	//	Weather temperature
END_VAR
VAR_INPUT CONSTANT
	BuildAlm				: FB_BA_BuildingAlarms;
	BuildMode				: FB_BA_BuildingMode;	
	WthParam				: FB_BA_WeatherParameter;
END_VAR
VAR
END_VAR
VAR // added by the converter: edge detectors and wires of the graphical bodies
    _s1 : ST_BA_GeneralSettings;
END_VAR

SUPER^(); // FB_BA_View
BuildAlm(); // FB_BA_BuildingAlarms
BuildMode(); // FB_BA_BuildingMode
WthParam(fTWth := fTWth); // FB_BA_WeatherParameter
// compose _s1 : ST_BA_GeneralSettings
_s1.fFrostProtectionSetpoint := WthParam.fSpFrstProtec;
_s1.fTWthLowLimit := WthParam.fTWthLowLimit;
_s1.bTWthLowLimit := WthParam.bTWthLowLimit;
_s1.fTWthDamped := WthParam.fTWthDamped;
_s1.bTWthDampedLowLimit := WthParam.bTWthDampedLowLimit;
_s1.fTWth := fTWth;
Site.stGeneralSettings := _s1;

METHOD FB_init : BOOL
VAR_INPUT
	bInitRetains : BOOL; // if TRUE, the retain variables are initialized (warm start / cold start)
	bInCopyCode : BOOL;  // if TRUE, the instance afterwards gets moved into the copy code (online change)
END_VAR
BuildAlm.iParent			:= THIS^;	
BuildAlm.iLabel				:= LblCtl_BuildingAlarms;
BuildAlm.eDPADMode			:= E_BA_DPADMode.eInclude;
                        
BuildMode.iParent			:= THIS^;	
BuildMode.iLabel			:= LblCtl_BuildingMode;
BuildMode.eDPADMode			:= E_BA_DPADMode.eInclude;

WthParam.iParent			:= THIS^;
WthParam.iLabel				:= LblCtl_WeatherParameters;
WthParam.eDPADMode			:= E_BA_DPADMode.eInclude;
END_METHOD

END_FUNCTION_BLOCK

// ---- Templates/POUs/Trade/BuildingAutomation/GlobalEventsAndSettings/FB_BA_BuildingAlarms.TcPOU
{region '#Template'}
	{attribute 'Version' := '5.0.0.0'}
	{attribute 'Tags' := '"LCID": "1031", "Text": "Gebäudeautomation, Betriebsarten"'}
	{attribute 'Tags' := '"LCID": "1033", "Text": "Building automation, Operating modes"'}
	{attribute 'Using' := '"Type": "Template", "URI": "BA2_Param"'}
	{attribute 'Using' := '"Type": "Template", "URI": "Site"'}		 
	{attribute 'Using' := '"Type": "Template", "URI": "EC_ID"'}
	{attribute 'Using' := '"Type": "Template", "URI": "ST_BA_BuildingAlarms"'}
	{attribute 'Description' := '"LCID": "1031", "Text": "Gebäude Betriebsarten"'}
	{attribute 'Description' := '"LCID": "1033", "Text": "Building operating modes"'}
{endregion}
FUNCTION_BLOCK FB_BA_BuildingAlarms EXTENDS FB_BA_View
VAR_INPUT CONSTANT
	FireAlert			: FB_BA_BI_Raw;                      
	Bgly				: FB_BA_BI_Raw;
	CentSwiOff			: FB_BA_BV_Op;
END_VAR
VAR // added by the converter: edge detectors and wires of the graphical bodies
    _s1 : ST_BA_BuildingAlarms;
END_VAR

SUPER^(); // FB_BA_View
FireAlert(); // FB_BA_BI_Raw
Bgly(); // FB_BA_BI_Raw
CentSwiOff(); // FB_BA_Bv_OP
// compose _s1 : ST_BA_BuildingAlarms
_s1.bBurglary := Bgly.bPresentValue;
_s1.bFireAlert := FireAlert.bPresentValue;
_s1.bCentralOff := CentSwiOff.bPresentValue;
_s1.bForcedVentilation := FALSE;
_s1.bSmokeExtraction := FALSE;
Site.stBuildingAlarms := _s1;

METHOD FB_init : BOOL
VAR_INPUT
	bInitRetains : BOOL; // if TRUE, the retain variables are initialized (warm start / cold start)
	bInCopyCode : BOOL;  // if TRUE, the instance afterwards gets moved into the copy code (online change)
END_VAR
FireAlert.iParent						:= THIS^;
FireAlert.iLabel						:= LblCtl_FireAlert;
FireAlert.bEnOutOfService				:= FALSE;
FireAlert.ePolarity						:= E_BA_Polarity.eReverse;
FireAlert.sActiveText 					:= txtEvent_Alert;
FireAlert.sInactiveText 				:= txtEvent_Normal;
FireAlert.nStateChangeCount				:= 0;
FireAlert.nActiveTimeElapsed			:= 0;
FireAlert.nEventClassID					:= EC_ID.NC10;
FireAlert.stTimeDelay.nToNormal			:= BA2_Param.nDefTimeDelay_ToNormal;
FireAlert.stTimeDelay.nToAbnormal		:= BA2_Param.nDefTimeDelay_ToAbnormal;
FireAlert.bAlarmValue					:= TRUE;
FireAlert.bAcknowledgeRm				:= FALSE;	
FireAlert.aEventTransitionText[1]		:= txtEvent_Alert;
FireAlert.aEventTransitionText[2]		:= txtEvent_None;
FireAlert.aEventTransitionText[3]		:= txtEvent_Normal;
FireAlert.bEventDetectionEnable			:= TRUE;

FireAlert.eEnPlantLock					:= E_BA_LockPriority.eNoLock;	

Bgly.iParent							:= THIS^;
Bgly.iLabel								:= LblCtl_Burglary;
Bgly.bEnOutOfService					:= FALSE;
Bgly.ePolarity							:= E_BA_Polarity.eReverse;
Bgly.sActiveText 						:= txtEvent_Alert;
Bgly.sInactiveText 						:= txtEvent_Normal;
Bgly.nStateChangeCount					:= 0;
Bgly.nActiveTimeElapsed					:= 0;
Bgly.nEventClassID						:= EC_ID.NC10;
Bgly.stTimeDelay.nToNormal				:= BA2_Param.nDefTimeDelay_ToNormal;
Bgly.stTimeDelay.nToAbnormal			:= BA2_Param.nDefTimeDelay_ToAbnormal;
Bgly.bAlarmValue						:= TRUE;
Bgly.bAcknowledgeRm						:= FALSE;	
Bgly.aEventTransitionText[1]			:= txtEvent_Alert;
Bgly.aEventTransitionText[2]			:= txtEvent_None;
Bgly.aEventTransitionText[3]			:= txtEvent_Normal; 
Bgly.bEventDetectionEnable				:= TRUE;

Bgly.eEnPlantLock						:= E_BA_LockPriority.eNoLock;	
                       	
CentSwiOff.iParent						:= THIS^;
CentSwiOff.iLabel						:= LblCtl_CentralSwitchOff;
CentSwiOff.sInactiveText				:= txtEvent_Off;
CentSwiOff.sActiveText					:= txtEvent_On;
CentSwiOff.bValueRm						:= FALSE;
CentSwiOff.eToggleMode					:= E_BA_ToggleMode.ePushButton;
END_METHOD

END_FUNCTION_BLOCK

// ---- Templates/POUs/Trade/BuildingAutomation/GlobalEventsAndSettings/FB_BA_BuildingMode.TcPOU
{region '#Template'}
	{attribute 'Version' := '5.0.0.0'}
	{attribute 'Tags' := '"LCID": "1031", "Text": "Gebäudeautomation, Building, Operating mode"'}
	{attribute 'Tags' := '"LCID": "1033", "Text": "Building automation, Building, Operating mode"'}
	{attribute 'Using' := '"Type": "Template", "URI": "Site"'}		 
	{attribute 'Using' := '"Type": "Template", "URI": "E_BA_BuildingMode"'}		 
	{attribute 'Description' := '"LCID": "1031", "Text": "Gebäude Betriebsart"'}
	{attribute 'Description' := '"LCID": "1033", "Text": "Building operating mode"'}
{endregion}
FUNCTION_BLOCK FB_BA_BuildingMode EXTENDS FB_BA_View
VAR_INPUT CONSTANT
	OpModMan					: FB_BA_MV_Op;
	OpModPr						: FB_BA_MV_Op;
	Sched						: FB_BA_SchedM;
END_VAR
VAR	
	DeMuxManMod					: FB_BA_DMUX_B04;		
	DeMuxSched					: FB_BA_DMUX_B04;		
	PrioSwi						: FB_BA_PrioSwi_UDI08;	
END_VAR

SUPER^(); // FB_BA_View
OpModMan(); // FB_BA_MV_Op
Sched(); // FB_BA_SchedM
DeMuxManMod(bEn := TRUE, nSel := OpModMan.nPresentValue, bIn := TRUE); // FB_BA_DMUX_B04
DeMuxSched(bEn := TRUE, nSel := Sched.nPresentValue, bIn := TRUE); // FB_BA_DMUX_B04
PrioSwi(
    bEn01 := DeMuxManMod.bQ02,
    nVal01 := E_BA_BuildingMode.eDefault,
    bEn02 := DeMuxManMod.bQ03,
    nVal02 := E_BA_BuildingMode.eNightWatch,
    bEn03 := DeMuxManMod.bQ04,
    nVal03 := E_BA_BuildingMode.eCleaning,
    bEn04 := FALSE,
    bEn05 := DeMuxSched.bQ01,
    nVal05 := E_BA_BuildingMode.eDefault,
    bEn06 := DeMuxSched.bQ02,
    nVal06 := E_BA_BuildingMode.eNightWatch,
    bEn07 := DeMuxSched.bQ03,
    nVal07 := E_BA_BuildingMode.eCleaning,
    bEn08 := FALSE); // FB_BA_PrioSwi_UDI08
OpModPr(nValuePgm := PrioSwi.nVal); // FB_BA_MV_Op
Site.eBuildingMode := PrioSwi.nVal;

METHOD FB_init : BOOL
VAR_INPUT
	bInitRetains : BOOL; // if TRUE, the retain variables are initialized (warm start / cold start)
	bInCopyCode : BOOL;  // if TRUE, the instance afterwards gets moved into the copy code (online change)
END_VAR
OpModMan.iParent		:= THIS^;
OpModMan.iLabel			:= LblCtl_BuildingModeManual;
OpModMan.aStateText[1]	:= txtEvent_Auto;
OpModMan.aStateText[2]	:= txtEvent_Default;
OpModMan.aStateText[3]	:= txtEvent_Nightwatch;
OpModMan.aStateText[4]	:= txtEvent_Cleaning;
OpModMan.nValueRm		:= 1;

OpModPr.iParent			:= THIS^;
OpModPr.iLabel			:= LblCtl_BuildingModeActual;	
OpModPr.aStateText[1]	:= txtEvent_Default;
OpModPr.aStateText[2]	:= txtEvent_Nightwatch;
OpModPr.aStateText[3]	:= txtEvent_Cleaning;
OpModPr.nValueRm		:= 1; 		
                        
Sched.iParent			:= THIS^;	
Sched.iLabel			:= LblCtl_BuildingModeSched;	
Sched.aStateText[1]		:= txtEvent_Default;
Sched.aStateText[2]		:= txtEvent_Nightwatch;
Sched.aStateText[3]		:= txtEvent_Cleaning;
Sched.nPredictTime		:= 0;


Sched.aWeek		:= F_BA_SchedWeekly4xM(E_BA_WeekDay.eMonday, E_BA_WeekDay.eFriday, T#0H, E_BA_BuildingMode.eNightWatch, T#6H, E_BA_BuildingMode.eDefault, T#19H, E_BA_BuildingMode.eCleaning, T#20H, E_BA_BuildingMode.eNightWatch);

